KUKA KRL program: MyProgram_191().src

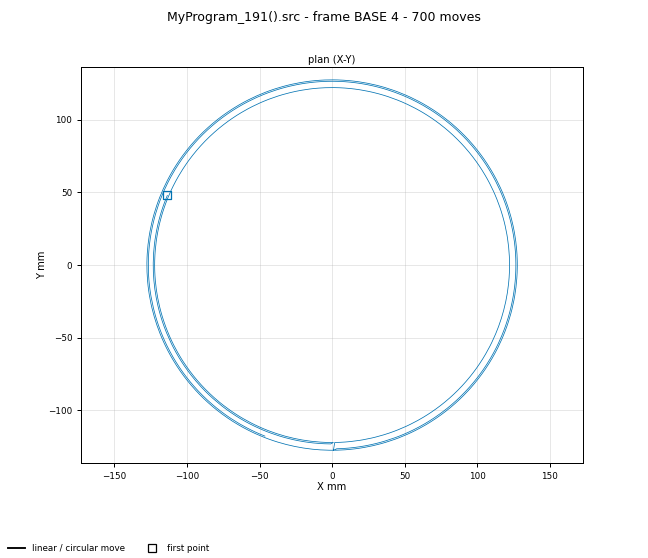
[picture p0: tool path of MyProgram_191().src in frame BASE 4, 700 of 700 moves have a stored position in this frame; points joined in program order, loops and branches not executed]
&ACCESS RVP
&REL 1
&PARAM TEMPLATE = C:\KRC\Roboter\Template\vorgabe
&PARAM EDITMASK = *
DEF MyProgram_191()
; ---- Setting reference (Base) ----
$BASE = BASE_DATA[4]

; --------------------------
; ---- Setting tool (TCP) ----
$TOOL = TOOL_DATA[3]
; --------------------------

$VEL.CP = VEL_APROX_PRINT
Startdeposition()
$VEL.CP = VEL_PRINT
LIN {X -113.4915,Y 47.9515,Z 138,A 153.5773,B 24.7784,C -1.6301,E1 24.6806,E2 292.6518} C_DIS
LIN {X -115.3064,Y 43.4036,Z 138,A 155.8653,B 24.7788,C -1.6235,E1 24.6783,E2 290.3668} C_DIS
LIN {X -116.411,Y 40.3471,Z 138,A 157.2234,B 24.7795,C -1.6121,E1 24.677,E2 289.0283} C_DIS
LIN {X -117.3905,Y 37.402,Z 138,A 158.8202,B 24.7794,C -1.6142,E1 24.6756,E2 287.4173} C_DIS
LIN {X -118.292,Y 34.4452,Z 138,A 160.3339,B 24.7794,C -1.6129,E1 24.6744,E2 285.8979} C_DIS
LIN {X -119.418,Y 30.3113,Z 138,A 162.2284,B 24.7801,C -1.6022,E1 24.6731,E2 284.0179} C_DIS
LIN {X -120.0632,Y 27.6462,Z 138,A 163.4846,B 24.7804,C -1.5973,E1 24.6723,E2 282.7662} C_DIS
LIN {X -120.9925,Y 23.2438,Z 138,A 165.6644,B 24.7806,C -1.5943,E1 24.6711,E2 280.5806} C_DIS
LIN {X -121.544,Y 20.1626,Z 138,A 167.1796,B 24.7806,C -1.5921,E1 24.6703,E2 279.0614} C_DIS
LIN {X -121.9177,Y 17.7672,Z 138,A 168.6693,B 24.78,C -1.6043,E1 24.6697,E2 277.5336} C_DIS
LIN {X -122.3545,Y 14.4523,Z 138,A 169.8773,B 24.7812,C -1.584,E1 24.6693,E2 276.3671} C_DIS
LIN {X -122.9178,Y 8.4272,Z 138,A 172.7848,B 24.7815,C -1.5788,E1 24.6687,E2 273.4544} C_DIS
LIN {X -123.1978,Y 1.4687,Z 138,A 176.8893,B 24.7798,C -1.6064,E1 24.6684,E2 269.2588} C_DIS
LIN {X -123.123,Y -4.5086,Z 138,A 178.5455,B 24.7833,C -1.5478,E1 24.6684,E2 267.7331} C_DIS
LIN {X -122.7454,Y -10.6368,Z 138,A -178.1412,B 24.7827,C -1.5585,E1 24.6691,E2 264.3741} C_DIS
LIN {X -122.0579,Y -16.7856,Z 138,A -175.5309,B 24.7839,C -1.5375,E1 24.67,E2 261.7985} C_DIS
LIN {X -121.0796,Y -22.7885,Z 138,A -172.5431,B 24.784,C -1.5354,E1 24.6714,E2 258.7978} C_DIS
LIN {X -120.0299,Y -27.7922,Z 138,A -170.1361,B 24.7844,C -1.5292,E1 24.6728,E2 256.3914} C_DIS
LIN {X -119.0923,Y -31.5671,Z 138,A -168.3681,B 24.7848,C -1.5218,E1 24.674,E2 254.6308} C_DIS
LIN {X -118.1261,Y -35.0118,Z 138,A -166.593,B 24.7848,C -1.5215,E1 24.6754,E2 252.8459} C_DIS
LIN {X -116.8426,Y -39.0802,Z 138,A -164.6565,B 24.7853,C -1.5134,E1 24.6771,E2 250.9178} C_DIS
LIN {X -115.6373,Y -42.5202,Z 138,A -163.0507,B 24.7858,C -1.5043,E1 24.6786,E2 249.3246} C_DIS
LIN {X -114.0487,Y -46.6116,Z 138,A -160.8655,B 24.7858,C -1.5046,E1 24.6809,E2 247.1262} C_DIS
LIN {X -110.5691,Y -54.3497,Z 138,A -156.9917,B 24.7866,C -1.49,E1 24.6854,E2 243.2662} C_DIS
LIN {X -109.2872,Y -56.8848,Z 138,A -155.6817,B 24.7869,C -1.4858,E1 24.687,E2 241.9592} C_DIS
LIN {X -107.5667,Y -60.078,Z 138,A -153.8305,B 24.7867,C -1.4884,E1 24.6895,E2 240.0919} C_DIS
LIN {X -105.3974,Y -63.8062,Z 138,A -152.0984,B 24.7877,C -1.4708,E1 24.692,E2 238.393} C_DIS
LIN {X -103.7402,Y -66.4666,Z 138,A -150.4231,B 24.7874,C -1.4766,E1 24.6945,E2 236.6952} C_DIS
LIN {X -101.5509,Y -69.7657,Z 138,A -148.5357,B 24.7875,C -1.4739,E1 24.6974,E2 234.8047} C_DIS
LIN {X -99.0053,Y -73.3341,Z 138,A -146.4687,B 24.7878,C -1.4701,E1 24.7008,E2 232.7369} C_DIS
LIN {X -96.9671,Y -76.0082,Z 138,A -144.6849,B 24.7874,C -1.4762,E1 24.7039,E2 230.93} C_DIS
LIN {X -93.5662,Y -80.158,Z 138,A -141.7973,B 24.7868,C -1.4881,E1 24.7093,E2 228.0006} C_DIS
LIN {X -90.2518,Y -83.8717,Z 138,A -140.0763,B 24.7885,C -1.4559,E1 24.7124,E2 226.3491} C_DIS
LIN {X -87.3058,Y -86.9342,Z 138,A -138.1334,B 24.7889,C -1.45,E1 24.7161,E2 224.4117} C_DIS
LIN {X -85.0375,Y -89.1542,Z 138,A -136.2104,B 24.7879,C -1.4673,E1 24.7201,E2 222.4395} C_DIS
LIN {X -82.0921,Y -91.8735,Z 138,A -135.1222,B 24.7901,C -1.4282,E1 24.7222,E2 221.4404} C_DIS
LIN {X -75.7976,Y -97.1325,Z 138,A -130.8704,B 24.7894,C -1.4406,E1 24.7315,E2 217.1426} C_DIS
LIN {X -72.8597,Y -99.3545,Z 138,A -129.1934,B 24.7896,C -1.4359,E1 24.7352,E2 215.4709} C_DIS
LIN {X -70.0805,Y -101.3345,Z 138,A -127.5112,B 24.7896,C -1.4376,E1 24.7391,E2 213.7788} C_DIS
LIN {X -66.1672,Y -103.9319,Z 138,A -125.6448,B 24.7905,C -1.4195,E1 24.7433,E2 211.9495} C_DIS
LIN {X -63.3912,Y -105.6482,Z 138,A -123.8429,B 24.7899,C -1.4303,E1 24.7477,E2 210.1162} C_DIS
LIN {X -59.6375,Y -107.811,Z 138,A -122.016,B 24.7906,C -1.4188,E1 24.7521,E2 208.3115} C_DIS
LIN {X -56.4456,Y -109.5155,Z 138,A -120.1657,B 24.7903,C -1.4243,E1 24.7567,E2 206.4429} C_DIS
LIN {X -53.2178,Y -111.1182,Z 138,A -118.5914,B 24.7906,C -1.4176,E1 24.7606,E2 204.8805} C_DIS
LIN {X -50.3384,Y -112.4519,Z 138,A -117.31,B 24.7912,C -1.4069,E1 24.7638,E2 203.6216} C_DIS
LIN {X -47.6999,Y -113.5965,Z 138,A -115.7642,B 24.7908,C -1.4151,E1 24.7679,E2 202.0525} C_DIS
LIN {X -45.0765,Y -114.6636,Z 138,A -114.595,B 24.7912,C -1.4069,E1 24.7709,E2 200.9003} C_DIS
LIN {X -41.9523,Y -115.8423,Z 138,A -113.0237,B 24.7912,C -1.4063,E1 24.775,E2 199.3272} C_DIS
LIN {X -39.061,Y -116.8489,Z 138,A -111.458,B 24.7909,C -1.4117,E1 24.7791,E2 197.7455} C_DIS
LIN {X -36.1486,Y -117.7825,Z 138,A -109.6372,B 24.79,C -1.4294,E1 24.7841,E2 195.8793} C_DIS
LIN {X -32.6362,Y -118.805,Z 138,A -108.2069,B 24.7907,C -1.4154,E1 24.7879,E2 194.48} C_DIS
LIN {X -26.8313,Y -120.2494,Z 138,A -105.5859,B 24.7912,C -1.4063,E1 24.795,E2 191.8771} C_DIS
LIN {X -23.219,Y -120.9973,Z 138,A -103.7988,B 24.7911,C -1.409,E1 24.7999,E2 190.0816} C_DIS
LIN {X -19.2814,Y -121.6877,Z 138,A -101.9432,B 24.7911,C -1.4083,E1 24.805,E2 188.226} C_DIS
LIN {X -16.1409,Y -122.1432,Z 138,A -100.6058,B 24.7915,C -1.4014,E1 24.8086,E2 186.904} C_DIS
LIN {X -13.0646,Y -122.5105,Z 138,A -98.9585,B 24.791,C -1.411,E1 24.8133,E2 185.2327} C_DIS
LIN {X -8.9867,Y -122.8769,Z 138,A -97.1257,B 24.7912,C -1.4075,E1 24.8184,E2 183.4074} C_DIS
LIN {X -5.1763,Y -123.097,Z 138,A -95.2835,B 24.791,C -1.4109,E1 24.8235,E2 181.5568} C_DIS
LIN {X -0.9339,Y -123.2019,Z 138,A -93.3832,B 24.7912,C -1.4077,E1 24.8288,E2 179.6639} C_DIS
LIN {X -0.9339,Y -123.2019,Z 138,A -93.3832,B 24.7912,C -1.4077,E1 24.8288,E2 179.6639} C_DIS
Enddeposition()
LIN {X 0.852,Y -122.218,Z 138,A -92.7365,B 24.3643,C -1.3273,E1 24.3999,E2 179.1497} C_DIS
Startdeposition()
$VEL.CP = VEL_PRINT
LIN {X -1.1747,Y -122.2187,Z 138,A -94.1532,B 24.3654,C -1.3055,E1 24.3958,E2 180.6191} C_DIS
LIN {X -4.4974,Y -122.1408,Z 138,A -95.7044,B 24.3654,C -1.3056,E1 24.3915,E2 182.1703} C_DIS
LIN {X -7.8683,Y -121.9703,Z 138,A -97.3656,B 24.3656,C -1.302,E1 24.3868,E2 183.8409} C_DIS
LIN {X -11.9845,Y -121.6346,Z 138,A -99.14,B 24.3652,C -1.3095,E1 24.3819,E2 185.598} C_DIS
LIN {X -14.6363,Y -121.3438,Z 138,A -100.3954,B 24.3652,C -1.3095,E1 24.3785,E2 186.8543} C_DIS
LIN {X -17.9306,Y -120.9025,Z 138,A -101.9314,B 24.3652,C -1.3108,E1 24.3742,E2 188.3883} C_DIS
LIN {X -20.5158,Y -120.4897,Z 138,A -103.2501,B 24.3654,C -1.307,E1 24.3706,E2 189.7174} C_DIS
LIN {X -23.5259,Y -119.939,Z 138,A -104.6142,B 24.3652,C -1.3108,E1 24.3668,E2 191.0739} C_DIS
LIN {X -26.0749,Y -119.4096,Z 138,A -105.9945,B 24.3655,C -1.3041,E1 24.363,E2 192.4721} C_DIS
LIN {X -29.708,Y -118.5582,Z 138,A -107.5972,B 24.3651,C -1.3117,E1 24.3587,E2 194.0587} C_DIS
LIN {X -32.2815,Y -117.8847,Z 138,A -108.8072,B 24.365,C -1.3141,E1 24.3555,E2 195.2647} C_DIS
LIN {X -35.4897,Y -116.9573,Z 138,A -110.2924,B 24.3648,C -1.3188,E1 24.3515,E2 196.7409} C_DIS
LIN {X -38.3454,Y -116.0524,Z 138,A -111.8191,B 24.365,C -1.3144,E1 24.3474,E2 198.2812} C_DIS
LIN {X -40.8707,Y -115.1886,Z 138,A -113.1758,B 24.3652,C -1.3108,E1 24.3438,E2 199.6495} C_DIS
LIN {X -43.6803,Y -114.1529,Z 138,A -114.5842,B 24.3652,C -1.3119,E1 24.3401,E2 201.0582} C_DIS
LIN {X -47.071,Y -112.7952,Z 138,A -116.2889,B 24.365,C -1.314,E1 24.3357,E2 202.7616} C_DIS
LIN {X -50.12,Y -111.474,Z 138,A -117.8196,B 24.3649,C -1.3169,E1 24.3318,E2 204.2891} C_DIS
LIN {X -53.3298,Y -109.9766,Z 138,A -119.4295,B 24.3646,C -1.3211,E1 24.3278,E2 205.893} C_DIS
LIN {X -56.0053,Y -108.6379,Z 138,A -120.8359,B 24.3646,C -1.3227,E1 24.3243,E2 207.2993} C_DIS
LIN {X -58.9088,Y -107.0922,Z 138,A -122.3786,B 24.3645,C -1.3248,E1 24.3205,E2 208.8415} C_DIS
LIN {X -61.2575,Y -105.7657,Z 138,A -123.7021,B 24.3645,C -1.324,E1 24.3173,E2 210.171} C_DIS
LIN {X -63.829,Y -104.234,Z 138,A -125.0526,B 24.3643,C -1.3284,E1 24.314,E2 211.515} C_DIS
LIN {X -66.6538,Y -102.4507,Z 138,A -126.6798,B 24.3643,C -1.3282,E1 24.3102,E2 213.1482} C_DIS
LIN {X -70.1137,Y -100.1153,Z 138,A -128.5919,B 24.364,C -1.3334,E1 24.3058,E2 215.0542} C_DIS
LIN {X -72.5492,Y -98.3643,Z 138,A -130.0014,B 24.3639,C -1.3357,E1 24.3026,E2 216.4632} C_DIS
LIN {X -74.9796,Y -96.5243,Z 138,A -131.4908,B 24.3639,C -1.3357,E1 24.2993,E2 217.9583} C_DIS
LIN {X -77.7047,Y -94.3448,Z 138,A -133.2287,B 24.3639,C -1.3342,E1 24.2955,E2 219.7062} C_DIS
LIN {X -81.0903,Y -91.4508,Z 138,A -135.2943,B 24.3637,C -1.3393,E1 24.2912,E2 221.7678} C_DIS
LIN {X -84.2804,Y -88.5197,Z 138,A -137.3634,B 24.3636,C -1.3419,E1 24.287,E2 223.8394} C_DIS
LIN {X -87.3611,Y -85.4805,Z 138,A -139.2827,B 24.3631,C -1.351,E1 24.2832,E2 225.7449} C_DIS
LIN {X -89.9719,Y -82.728,Z 138,A -141.1255,B 24.3631,C -1.3522,E1 24.2797,E2 227.5931} C_DIS
LIN {X -92.9374,Y -79.3826,Z 138,A -143.1994,B 24.3627,C -1.3579,E1 24.2759,E2 229.6626} C_DIS
LIN {X -95.4175,Y -76.3838,Z 138,A -145.1405,B 24.3627,C -1.3573,E1 24.2724,E2 231.6145} C_DIS
LIN {X -98.1723,Y -72.8088,Z 138,A -147.1088,B 24.3622,C -1.3688,E1 24.2691,E2 233.5645} C_DIS
LIN {X -100.0245,Y -70.2427,Z 138,A -148.764,B 24.3624,C -1.3652,E1 24.2664,E2 235.2367} C_DIS
LIN {X -102.4504,Y -66.6543,Z 138,A -150.5579,B 24.3615,C -1.3806,E1 24.2637,E2 237.0023} C_DIS
LIN {X -104.0513,Y -64.1269,Z 138,A -152.1971,B 24.3619,C -1.3742,E1 24.2612,E2 238.6658} C_DIS
LIN {X -106.3494,Y -60.2395,Z 138,A -154.1332,B 24.3612,C -1.3876,E1 24.2586,E2 240.5795} C_DIS
LIN {X -107.6369,Y -57.9065,Z 138,A -155.5184,B 24.3612,C -1.3853,E1 24.2567,E2 241.9778} C_DIS
LIN {X -109.0137,Y -55.2671,Z 138,A -156.8887,B 24.361,C -1.3903,E1 24.2549,E2 243.3435} C_DIS
LIN {X -110.5038,Y -52.2262,Z 138,A -158.4413,B 24.3607,C -1.3963,E1 24.2531,E2 244.8902} C_DIS
LIN {X -111.8809,Y -49.2103,Z 138,A -160.2288,B 24.361,C -1.3909,E1 24.251,E2 246.701} C_DIS
LIN {X -113.483,Y -45.3887,Z 138,A -161.957,B 24.3602,C -1.4057,E1 24.2492,E2 248.403} C_DIS
LIN {X -114.5655,Y -42.5825,Z 138,A -163.4393,B 24.3602,C -1.4068,E1 24.2477,E2 249.8911} C_DIS
LIN {X -115.9501,Y -38.6526,Z 138,A -165.4017,B 24.3598,C -1.4123,E1 24.2459,E2 251.8516} C_DIS
LIN {X -116.9523,Y -35.5062,Z 138,A -166.9,B 24.3595,C -1.4191,E1 24.2447,E2 253.3422} C_DIS
LIN {X -117.9764,Y -31.9412,Z 138,A -168.7779,B 24.3595,C -1.4186,E1 24.2433,E2 255.2325} C_DIS
LIN {X -118.839,Y -28.5616,Z 138,A -170.2955,B 24.3589,C -1.4286,E1 24.2423,E2 256.7347} C_DIS
LIN {X -119.5751,Y -25.3083,Z 138,A -171.8644,B 24.3587,C -1.4333,E1 24.2413,E2 258.3017} C_DIS
LIN {X -120.0655,Y -22.8641,Z 138,A -173.0773,B 24.3586,C -1.4351,E1 24.2407,E2 259.5175} C_DIS
LIN {X -120.6223,Y -19.7208,Z 138,A -174.5459,B 24.3583,C -1.441,E1 24.24,E2 260.9807} C_DIS
LIN {X -121.0678,Y -16.7739,Z 138,A -176.0325,B 24.3583,C -1.4417,E1 24.2394,E2 262.4747} C_DIS
LIN {X -121.4911,Y -13.3604,Z 138,A -177.4882,B 24.3576,C -1.4535,E1 24.2389,E2 263.9106} C_DIS
LIN {X -121.7522,Y -10.7287,Z 138,A -178.9175,B 24.3578,C -1.4496,E1 24.2386,E2 265.3584} C_DIS
LIN {X -121.9947,Y -7.4711,Z 138,A 179.6289,B 24.3573,C -1.4578,E1 24.2383,E2 266.801} C_DIS
LIN {X -122.1625,Y -3.8853,Z 138,A 177.7938,B 24.3573,C -1.4568,E1 24.2381,E2 268.6497} C_DIS
LIN {X -122.2263,Y -0.1231,Z 138,A 176.0896,B 24.3569,C -1.465,E1 24.2381,E2 270.3444} C_DIS
LIN {X -122.1899,Y 2.8995,Z 138,A 174.6031,B 24.3569,C -1.4668,E1 24.2381,E2 271.8359} C_DIS
LIN {X -122.0207,Y 7.0487,Z 138,A 172.7178,B 24.3563,C -1.4757,E1 24.2384,E2 273.7111} C_DIS
LIN {X -121.8016,Y 10.1449,Z 138,A 171.2313,B 24.3561,C -1.4792,E1 24.2387,E2 275.1983} C_DIS
LIN {X -121.4789,Y 13.4743,Z 138,A 169.764,B 24.3556,C -1.4885,E1 24.2391,E2 276.652} C_DIS
LIN {X -121.1532,Y 16.1393,Z 138,A 168.4248,B 24.3556,C -1.4892,E1 24.2396,E2 277.9977} C_DIS
LIN {X -120.599,Y 19.8602,Z 138,A 166.5949,B 24.3554,C -1.4922,E1 24.2404,E2 279.8315} C_DIS
LIN {X -119.9418,Y 23.5111,Z 138,A 164.9317,B 24.3549,C -1.5009,E1 24.2412,E2 281.4834} C_DIS
LIN {X -119.3249,Y 26.4675,Z 138,A 163.3914,B 24.3549,C -1.5003,E1 24.2421,E2 283.0346} C_DIS
LIN {X -118.5602,Y 29.6998,Z 138,A 161.7993,B 24.3547,C -1.5039,E1 24.2432,E2 284.6276} C_DIS
LIN {X -117.4803,Y 33.7233,Z 138,A 159.8547,B 24.3543,C -1.5104,E1 24.2446,E2 286.5679} C_DIS
LIN {X -116.6188,Y 36.5911,Z 138,A 158.4425,B 24.3541,C -1.5145,E1 24.2458,E2 287.9784} C_DIS
LIN {X -115.5784,Y 39.7513,Z 138,A 156.8856,B 24.3538,C -1.5196,E1 24.2472,E2 289.5321} C_DIS
LIN {X -114.3716,Y 43.1001,Z 138,A 155.1973,B 24.3535,C -1.524,E1 24.2488,E2 291.2195} C_DIS
LIN {X -113.0423,Y 46.4791,Z 138,A 153.48,B 24.3532,C -1.5286,E1 24.2506,E2 292.9354} C_DIS
LIN {X -111.8746,Y 49.2245,Z 138,A 152.0617,B 24.353,C -1.532,E1 24.2522,E2 294.3534} C_DIS
LIN {X -110.6278,Y 51.9657,Z 138,A 150.7478,B 24.3525,C -1.5404,E1 24.2537,E2 295.6543} C_DIS
LIN {X -109.3219,Y 54.6585,Z 138,A 149.3353,B 24.3523,C -1.5442,E1 24.2555,E2 297.0653} C_DIS
LIN {X -107.5634,Y 58.0433,Z 138,A 147.521,B 24.3521,C -1.5484,E1 24.2578,E2 298.8792} C_DIS
LIN {X -105.7031,Y 61.3657,Z 138,A 145.7038,B 24.3518,C -1.5523,E1 24.2603,E2 300.6967} C_DIS
LIN {X -104.2135,Y 63.8625,Z 138,A 144.4625,B 24.3513,C -1.5614,E1 24.2621,E2 301.9224} C_DIS
LIN {X -102.6967,Y 66.2749,Z 138,A 142.8668,B 24.3517,C -1.5542,E1 24.2645,E2 303.5438} C_DIS
LIN {X -100.1153,Y 70.1137,Z 138,A 140.8425,B 24.351,C -1.5664,E1 24.2677,E2 305.5489} C_DIS
LIN {X -98.3676,Y 72.5447,Z 138,A 139.3725,B 24.351,C -1.5674,E1 24.2701,E2 307.0236} C_DIS
LIN {X -95.8913,Y 75.7882,Z 138,A 137.3452,B 24.351,C -1.5678,E1 24.2736,E2 309.06} C_DIS
LIN {X -93.1416,Y 79.1423,Z 138,A 135.4038,B 24.3503,C -1.577,E1 24.277,E2 310.9882} C_DIS
LIN {X -90.5637,Y 82.0798,Z 138,A 133.4693,B 24.3503,C -1.5773,E1 24.2807,E2 312.9307} C_DIS
LIN {X -87.5282,Y 85.3101,Z 138,A 131.3586,B 24.3501,C -1.5811,E1 24.2847,E2 315.0416} C_DIS
LIN {X -84.2766,Y 88.5233,Z 138,A 129.2184,B 24.3498,C -1.5864,E1 24.289,E2 317.1782} C_DIS
LIN {X -81.09,Y 91.4512,Z 138,A 127.2157,B 24.3494,C -1.5922,E1 24.2932,E2 319.1749} C_DIS
LIN {X -78.0552,Y 94.0546,Z 138,A 125.3237,B 24.3492,C -1.5957,E1 24.2972,E2 321.066} C_DIS
LIN {X -74.6019,Y 96.8171,Z 138,A 123.2103,B 24.349,C -1.5984,E1 24.3018,E2 323.1806} C_DIS
LIN {X -71.6013,Y 99.0563,Z 138,A 121.6099,B 24.3484,C -1.6087,E1 24.3054,E2 324.7618} C_DIS
LIN {X -69.1523,Y 100.781,Z 138,A 120.1252,B 24.3484,C -1.6081,E1 24.3088,E2 326.2533} C_DIS
LIN {X -65.6572,Y 103.0926,Z 138,A 118.1515,B 24.3482,C -1.6115,E1 24.3134,E2 328.2253} C_DIS
LIN {X -62.8163,Y 104.8478,Z 138,A 116.7156,B 24.3477,C -1.62,E1 24.3168,E2 329.6451} C_DIS
LIN {X -60.2331,Y 106.3531,Z 138,A 115.2944,B 24.3476,C -1.6216,E1 24.3203,E2 331.0666} C_DIS
LIN {X -57.9016,Y 107.6396,Z 138,A 113.9157,B 24.3478,C -1.6181,E1 24.3237,E2 332.4578} C_DIS
LIN {X -54.9576,Y 109.1713,Z 138,A 112.4297,B 24.3475,C -1.6237,E1 24.3273,E2 333.9343} C_DIS
LIN {X -52.1843,Y 110.5239,Z 138,A 110.9805,B 24.3473,C -1.6259,E1 24.331,E2 335.3821} C_DIS
LIN {X -49.5255,Y 111.7399,Z 138,A 109.6064,B 24.3473,C -1.6278,E1 24.3345,E2 336.755} C_DIS
LIN {X -47.0747,Y 112.7936,Z 138,A 108.2983,B 24.3473,C -1.6272,E1 24.3379,E2 338.0678} C_DIS
LIN {X -43.5437,Y 114.2055,Z 138,A 106.3657,B 24.3475,C -1.623,E1 24.3429,E2 340.0147} C_DIS
LIN {X -39.8373,Y 115.5486,Z 138,A 104.7562,B 24.3467,C -1.6358,E1 24.3471,E2 341.5964} C_DIS
LIN {X -37.2178,Y 116.4185,Z 138,A 103.358,B 24.3469,C -1.6328,E1 24.3508,E2 343.0046} C_DIS
LIN {X -34.0409,Y 117.3872,Z 138,A 101.8572,B 24.3466,C -1.637,E1 24.3548,E2 344.4977} C_DIS
LIN {X -31.1552,Y 118.186,Z 138,A 100.4972,B 24.3464,C -1.6403,E1 24.3585,E2 345.8517} C_DIS
LIN {X -28.5721,Y 118.8365,Z 138,A 99.1492,B 24.3466,C -1.6372,E1 24.3621,E2 347.2093} C_DIS
LIN {X -25.0186,Y 119.6369,Z 138,A 97.3083,B 24.3469,C -1.6328,E1 24.3672,E2 349.0633} C_DIS
LIN {X -21.2072,Y 120.3696,Z 138,A 95.6706,B 24.3463,C -1.6422,E1 24.3716,E2 350.6798} C_DIS
LIN {X -18.2515,Y 120.8536,Z 138,A 94.2678,B 24.3463,C -1.6432,E1 24.3755,E2 352.0814} C_DIS
LIN {X -15.318,Y 121.2608,Z 138,A 92.7722,B 24.3465,C -1.6393,E1 24.3797,E2 353.5877} C_DIS
LIN {X -12.3074,Y 121.6036,Z 138,A 91.4293,B 24.3462,C -1.6435,E1 24.3834,E2 354.9211} C_DIS
LIN {X -8.9578,Y 121.8946,Z 138,A 89.8085,B 24.3462,C -1.6423,E1 24.3879,E2 356.5458} C_DIS
LIN {X -4.8186,Y 122.1283,Z 138,A 87.9232,B 24.3461,C -1.6455,E1 24.3931,E2 358.4236} C_DIS
LIN {X -1.8245,Y 122.2099,Z 138,A 86.4961,B 24.3461,C -1.6449,E1 24.3971,E2 359.8524} C_DIS
LIN {X 1.1685,Y 122.2188,Z 138,A 84.9591,B 24.3465,C -1.6391,E1 24.4015,E2 361.4034} C_DIS
LIN {X 5.2319,Y 122.1122,Z 138,A 83.0229,B 24.3465,C -1.6379,E1 24.4069,E2 363.342} C_DIS
LIN {X 8.669,Y 121.9156,Z 138,A 81.588,B 24.3461,C -1.6459,E1 24.4108,E2 364.7569} C_DIS
LIN {X 11.9806,Y 121.635,Z 138,A 80.0447,B 24.3461,C -1.6464,E1 24.4151,E2 366.298} C_DIS
LIN {X 15.5903,Y 121.2251,Z 138,A 78.2696,B 24.3463,C -1.6428,E1 24.42,E2 368.0805} C_DIS
LIN {X 19.4212,Y 120.6723,Z 138,A 76.5086,B 24.3461,C -1.6447,E1 24.4249,E2 369.8353} C_DIS
LIN {X 22.3721,Y 120.1595,Z 138,A 75.185,B 24.3459,C -1.6478,E1 24.4285,E2 371.1498} C_DIS
LIN {X 25.0145,Y 119.6377,Z 138,A 73.8644,B 24.3461,C -1.6446,E1 24.4321,E2 372.4765} C_DIS
LIN {X 28.1611,Y 118.9355,Z 138,A 72.171,B 24.3467,C -1.6354,E1 24.4368,E2 374.1897} C_DIS
LIN {X 32.2917,Y 117.8818,Z 138,A 70.3516,B 24.3463,C -1.6423,E1 24.4417,E2 375.9894} C_DIS
LIN {X 35.4859,Y 116.9585,Z 138,A 68.9156,B 24.346,C -1.6468,E1 24.4455,E2 377.412} C_DIS
LIN {X 38.6541,Y 115.9496,Z 138,A 67.1084,B 24.3468,C -1.6341,E1 24.4503,E2 379.2465} C_DIS
LIN {X 42.5823,Y 114.5656,Z 138,A 65.4196,B 24.3462,C -1.6445,E1 24.4547,E2 380.9067} C_DIS
LIN {X 45.0698,Y 113.6116,Z 138,A 63.8894,B 24.3471,C -1.6302,E1 24.4588,E2 382.468} C_DIS
LIN {X 48.3908,Y 112.2353,Z 138,A 62.3278,B 24.3468,C -1.6341,E1 24.4627,E2 384.0164} C_DIS
LIN {X 51.9751,Y 110.6235,Z 138,A 60.5174,B 24.3468,C -1.6333,E1 24.4673,E2 385.8238} C_DIS
LIN {X 54.6661,Y 109.3182,Z 138,A 59.1189,B 24.347,C -1.6317,E1 24.4708,E2 387.2223} C_DIS
LIN {X 57.3256,Y 107.9467,Z 138,A 57.6875,B 24.3472,C -1.6285,E1 24.4744,E2 388.6574} C_DIS
LIN {X 60.2381,Y 106.3503,Z 138,A 56.221,B 24.347,C -1.6305,E1 24.4779,E2 390.1146} C_DIS
LIN {X 62.8397,Y 104.8338,Z 138,A 54.7644,B 24.3473,C -1.6263,E1 24.4815,E2 391.5768} C_DIS
LIN {X 65.6974,Y 103.0668,Z 138,A 53.056,B 24.3478,C -1.6176,E1 24.4855,E2 393.3007} C_DIS
LIN {X 68.8222,Y 101.0074,Z 138,A 51.4364,B 24.3476,C -1.621,E1 24.4893,E2 394.9065} C_DIS
LIN {X 71.3331,Y 99.2499,Z 138,A 50.1139,B 24.3474,C -1.6239,E1 24.4923,E2 396.2172} C_DIS
LIN {X 74.0069,Y 97.2725,Z 138,A 48.3132,B 24.3483,C -1.6097,E1 24.4963,E2 398.0456} C_DIS
LIN {X 77.5317,Y 94.4868,Z 138,A 46.3116,B 24.3483,C -1.6107,E1 24.5007,E2 400.0371} C_DIS
LIN {X 80.2808,Y 92.1622,Z 138,A 44.6537,B 24.3483,C -1.6088,E1 24.5042,E2 401.693} C_DIS
LIN {X 83.1858,Y 89.5489,Z 138,A 42.7529,B 24.3488,C -1.6017,E1 24.5081,E2 403.6028} C_DIS
LIN {X 86.088,Y 86.7625,Z 138,A 40.861,B 24.3491,C -1.5974,E1 24.5119,E2 405.4971} C_DIS
LIN {X 89.0365,Y 83.7341,Z 138,A 38.891,B 24.3493,C -1.5936,E1 24.5157,E2 407.4677} C_DIS
LIN {X 91.559,Y 80.9679,Z 138,A 37.1512,B 24.3495,C -1.5903,E1 24.519,E2 409.2075} C_DIS
LIN {X 94.3821,Y 77.6597,Z 138,A 35.2027,B 24.3495,C -1.5897,E1 24.5224,E2 411.148} C_DIS
LIN {X 96.8164,Y 74.6028,Z 138,A 33.3331,B 24.35,C -1.5834,E1 24.5257,E2 413.0237} C_DIS
LIN {X 99.0689,Y 71.5838,Z 138,A 31.608,B 24.3501,C -1.581,E1 24.5285,E2 414.7463} C_DIS
LIN {X 101.4348,Y 68.1908,Z 138,A 29.6468,B 24.3505,C -1.5749,E1 24.5316,E2 416.7123} C_DIS
LIN {X 103.1672,Y 65.5402,Z 138,A 28.1069,B 24.3509,C -1.5683,E1 24.534,E2 418.2601} C_DIS
LIN {X 105.4236,Y 61.8444,Z 138,A 26.1818,B 24.3509,C -1.5679,E1 24.5367,E2 420.176} C_DIS
LIN {X 106.9194,Y 59.2208,Z 138,A 24.8348,B 24.3509,C -1.5673,E1 24.5386,E2 421.5173} C_DIS
LIN {X 108.489,Y 56.2929,Z 138,A 23.2787,B 24.3512,C -1.563,E1 24.5406,E2 423.0752} C_DIS
LIN {X 109.8352,Y 53.6181,Z 138,A 21.8856,B 24.3514,C -1.5596,E1 24.5423,E2 424.469} C_DIS
LIN {X 111.0995,Y 50.9457,Z 138,A 20.5469,B 24.3514,C -1.5579,E1 24.5439,E2 425.8044} C_DIS
LIN {X 112.1692,Y 48.5437,Z 138,A 19.2668,B 24.3519,C -1.552,E1 24.5453,E2 427.0914} C_DIS
LIN {X 113.4868,Y 45.3792,Z 138,A 17.6905,B 24.352,C -1.5488,E1 24.547,E2 428.6667} C_DIS
LIN {X 114.565,Y 42.5839,Z 138,A 16.3492,B 24.3521,C -1.5477,E1 24.5483,E2 430.003} C_DIS
LIN {X 115.5744,Y 39.7629,Z 138,A 14.9561,B 24.3523,C -1.544,E1 24.5496,E2 431.3969} C_DIS
LIN {X 116.4249,Y 37.198,Z 138,A 13.5879,B 24.3529,C -1.5352,E1 24.5508,E2 432.7783} C_DIS
LIN {X 117.3902,Y 34.0308,Z 138,A 11.9691,B 24.3533,C -1.5272,E1 24.5521,E2 434.4069} C_DIS
LIN {X 118.479,Y 30.0198,Z 138,A 10.1674,B 24.3533,C -1.5283,E1 24.5534,E2 436.1953} C_DIS
LIN {X 119.1774,Y 27.1152,Z 138,A 8.7309,B 24.3536,C -1.5221,E1 24.5543,E2 437.6381} C_DIS
LIN {X 119.8759,Y 23.8439,Z 138,A 7.2256,B 24.3537,C -1.5202,E1 24.5552,E2 439.139} C_DIS
LIN {X 120.3669,Y 21.2227,Z 138,A 5.9821,B 24.3539,C -1.5166,E1 24.5558,E2 440.3837} C_DIS
LIN {X 120.8017,Y 18.5867,Z 138,A 4.7116,B 24.3542,C -1.5117,E1 24.5563,E2 441.6583} C_DIS
LIN {X 121.3054,Y 14.9578,Z 138,A 3.0159,B 24.3545,C -1.5073,E1 24.557,E2 443.3544} C_DIS
LIN {X 121.6036,Y 12.3073,Z 138,A 1.7691,B 24.3547,C -1.5034,E1 24.5573,E2 444.603} C_DIS
LIN {X 121.8918,Y 8.9951,Z 138,A 0.3033,B 24.3547,C -1.5029,E1 24.5577,E2 446.061} C_DIS
LIN {X 122.0729,Y 6.0625,Z 138,A -1.1822,B 24.3553,C -1.4931,E1 24.5579,E2 447.561} C_DIS
LIN {X 122.2099,Y 1.827,Z 138,A -3.0667,B 24.3553,C -1.4917,E1 24.558,E2 449.4375} C_DIS
LIN {X 122.2153,Y -1.4969,Z 138,A -4.6683,B 24.3558,C -1.4844,E1 24.558,E2 451.0468} C_DIS
LIN {X 122.1283,Y -4.8191,Z 138,A -6.2088,B 24.356,C -1.4802,E1 24.5579,E2 452.588} C_DIS
LIN {X 121.9159,Y -8.6657,Z 138,A -8.0616,B 24.3565,C -1.472,E1 24.5576,E2 454.4494} C_DIS
LIN {X 121.5558,Y -12.7597,Z 138,A -9.9936,B 24.3569,C -1.4654,E1 24.557,E2 456.3854} C_DIS
LIN {X 121.156,Y -16.1174,Z 138,A -11.506,B 24.3569,C -1.4638,E1 24.5565,E2 457.8925} C_DIS
LIN {X 120.7332,Y -19.029,Z 138,A -12.8222,B 24.3571,C -1.4624,E1 24.556,E2 459.2041} C_DIS
LIN {X 120.1584,Y -22.3784,Z 138,A -14.3591,B 24.3571,C -1.46,E1 24.5552,E2 460.7377} C_DIS
LIN {X 119.6367,Y -25.0196,Z 138,A -15.6741,B 24.3576,C -1.4533,E1 24.5545,E2 462.0609} C_DIS
LIN {X 118.9142,Y -28.2497,Z 138,A -17.226,B 24.3579,C -1.4483,E1 24.5535,E2 463.6156} C_DIS
LIN {X 118.187,Y -31.1516,Z 138,A -18.4902,B 24.3577,C -1.4505,E1 24.5526,E2 464.8668} C_DIS
LIN {X 117.4819,Y -33.7176,Z 138,A -19.9614,B 24.3586,C -1.4356,E1 24.5515,E2 466.3655} C_DIS
LIN {X 116.6226,Y -36.579,Z 138,A -21.3566,B 24.3588,C -1.4314,E1 24.5504,E2 467.7627} C_DIS
LIN {X 115.5762,Y -39.7575,Z 138,A -22.6783,B 24.3584,C -1.4385,E1 24.5492,E2 469.0595} C_DIS
LIN {X 114.6008,Y -42.4884,Z 138,A -24.0658,B 24.3587,C -1.4329,E1 24.5479,E2 470.4526} C_DIS
LIN {X 113.6089,Y -45.0766,Z 138,A -25.4399,B 24.3591,C -1.4251,E1 24.5465,E2 471.8375} C_DIS
LIN {X 112.6264,Y -47.4751,Z 138,A -26.7235,B 24.3595,C -1.418,E1 24.5451,E2 473.131} C_DIS
LIN {X 111.1086,Y -50.9259,Z 138,A -28.2644,B 24.3592,C -1.4237,E1 24.5434,E2 474.6497} C_DIS
LIN {X 109.9776,Y -53.3277,Z 138,A -29.6473,B 24.3598,C -1.4131,E1 24.5417,E2 476.0504} C_DIS
LIN {X 108.6491,Y -55.9834,Z 138,A -31.033,B 24.36,C -1.4092,E1 24.5399,E2 477.4378} C_DIS
LIN {X 107.075,Y -58.9399,Z 138,A -32.5812,B 24.3602,C -1.4056,E1 24.5379,E2 478.9864} C_DIS
LIN {X 105.7622,Y -61.2636,Z 138,A -33.8873,B 24.3605,C -1.3992,E1 24.5361,E2 480.3009} C_DIS
LIN {X 103.7135,Y -64.6714,Z 138,A -35.7592,B 24.3609,C -1.3934,E1 24.5333,E2 482.177} C_DIS
LIN {X 101.4374,Y -68.187,Z 138,A -37.8095,B 24.3614,C -1.3836,E1 24.5302,E2 484.2405} C_DIS
LIN {X 99.2488,Y -71.3346,Z 138,A -39.4241,B 24.3612,C -1.3875,E1 24.5276,E2 485.8378} C_DIS
LIN {X 97.273,Y -74.0063,Z 138,A -41.0994,B 24.3617,C -1.3775,E1 24.5247,E2 487.5288} C_DIS
LIN {X 94.8419,Y -77.0972,Z 138,A -42.9286,B 24.3619,C -1.3732,E1 24.5215,E2 489.3596} C_DIS
LIN {X 92.163,Y -80.2798,Z 138,A -44.7745,B 24.3619,C -1.3732,E1 24.5182,E2 491.197} C_DIS
LIN {X 89.551,Y -83.1836,Z 138,A -46.6766,B 24.3624,C -1.365,E1 24.5146,E2 493.1102} C_DIS
LIN {X 86.5318,Y -86.3202,Z 138,A -48.6545,B 24.3624,C -1.363,E1 24.5108,E2 495.0842} C_DIS
LIN {X 83.7307,Y -89.0397,Z 138,A -50.5354,B 24.3628,C -1.3561,E1 24.5069,E2 496.9738} C_DIS
LIN {X 80.966,Y -91.5608,Z 138,A -52.2747,B 24.363,C -1.3527,E1 24.5033,E2 498.7141} C_DIS
LIN {X 77.6568,Y -94.3845,Z 138,A -54.2242,B 24.363,C -1.3523,E1 24.4992,E2 500.6567} C_DIS
LIN {X 74.6009,Y -96.8178,Z 138,A -56.1703,B 24.3635,C -1.3428,E1 24.4949,E2 502.6184} C_DIS
LIN {X 71.6009,Y -99.0566,Z 138,A -57.81,B 24.3635,C -1.3446,E1 24.4912,E2 504.2477} C_DIS
LIN {X 68.1881,Y -101.4367,Z 138,A -59.7848,B 24.3637,C -1.3395,E1 24.4866,E2 506.228} C_DIS
LIN {X 65.6646,Y -103.0879,Z 138,A -61.0446,B 24.3635,C -1.3441,E1 24.4837,E2 507.4725} C_DIS
LIN {X 62.8335,Y -104.8375,Z 138,A -62.8091,B 24.3641,C -1.3314,E1 24.4795,E2 509.262} C_DIS
LIN {X 59.0212,Y -107.03,Z 138,A -64.6958,B 24.3639,C -1.336,E1 24.4749,E2 511.1318} C_DIS
LIN {X 56.2496,Y -108.5118,Z 138,A -66.1484,B 24.3639,C -1.3344,E1 24.4713,E2 512.584} C_DIS
LIN {X 53.928,Y -109.6823,Z 138,A -67.4464,B 24.3643,C -1.3287,E1 24.468,E2 513.8923} C_DIS
LIN {X 50.888,Y -111.1262,Z 138,A -68.9691,B 24.3643,C -1.3287,E1 24.4642,E2 515.4107} C_DIS
LIN {X 48.1495,Y -112.3396,Z 138,A -70.3222,B 24.3643,C -1.3291,E1 24.4608,E2 516.7597} C_DIS
LIN {X 45.3817,Y -113.4859,Z 138,A -71.7661,B 24.3644,C -1.3252,E1 24.457,E2 518.2097} C_DIS
LIN {X 42.7791,Y -114.4919,Z 138,A -73.104,B 24.3646,C -1.322,E1 24.4535,E2 519.5524} C_DIS
LIN {X 39.3734,Y -115.7094,Z 138,A -74.9712,B 24.3651,C -1.3117,E1 24.4485,E2 521.4406} C_DIS
LIN {X 35.4629,Y -116.9655,Z 138,A -76.6286,B 24.3646,C -1.322,E1 24.4442,E2 523.0699} C_DIS
LIN {X 32.5932,Y -117.7975,Z 138,A -78.0746,B 24.3648,C -1.3183,E1 24.4403,E2 524.5223} C_DIS
LIN {X 30.022,Y -118.4785,Z 138,A -79.3196,B 24.3648,C -1.3171,E1 24.4369,E2 525.7683} C_DIS
LIN {X 27.1194,Y -119.1764,Z 138,A -80.7621,B 24.365,C -1.3137,E1 24.433,E2 527.2169} C_DIS
LIN {X 23.841,Y -119.8765,Z 138,A -82.2781,B 24.365,C -1.3149,E1 24.4288,E2 528.7281} C_DIS
LIN {X 21.2194,Y -120.3674,Z 138,A -83.4918,B 24.365,C -1.3156,E1 24.4255,E2 529.9387} C_DIS
LIN {X 18.6654,Y -120.7895,Z 138,A -84.8042,B 24.3652,C -1.3101,E1 24.4219,E2 531.2631} C_DIS
LIN {X 14.955,Y -121.3057,Z 138,A -86.51,B 24.3652,C -1.3113,E1 24.4171,E2 532.9646} C_DIS
LIN {X 12.3037,Y -121.604,Z 138,A -87.7649,B 24.3652,C -1.3104,E1 24.4137,E2 534.2208} C_DIS
LIN {X 8.9925,Y -121.892,Z 138,A -89.3062,B 24.3652,C -1.3104,E1 24.4094,E2 535.7612} C_DIS
LIN {X 5.7189,Y -122.0901,Z 138,A -90.9883,B 24.3656,C -1.3031,E1 24.4046,E2 537.4604} C_DIS
LIN {X 1.8206,Y -122.21,Z 138,A -92.6906,B 24.3653,C -1.3084,E1 24.3999,E2 539.1497} C_DIS
LIN {X 1.8206,Y -122.21,Z 138,A -92.6906,B 24.3653,C -1.3084,E1 24.3999,E2 539.1497} C_DIS
Enddeposition()
LIN {X 0.903,Y -127.5582,Z 139,A -92.8335,B 24.9653,C -1.3615,E1 25.0014,E2 539.248} C_DIS
Startdeposition()
$VEL.CP = VEL_PRINT
LIN {X -1.9731,Y -127.547,Z 139,A -94.4529,B 24.9661,C -1.3449,E1 24.9968,E2 540.9066} C_DIS
LIN {X -5.6447,Y -127.439,Z 139,A -96.0438,B 24.966,C -1.3476,E1 24.9924,E2 542.4915} C_DIS
LIN {X -8.0273,Y -127.3094,Z 139,A -97.1271,B 24.966,C -1.347,E1 24.9893,E2 543.5765} C_DIS
LIN {X -11.3552,Y -127.0572,Z 139,A -98.6178,B 24.966,C -1.3474,E1 24.9852,E2 545.0668} C_DIS
LIN {X -13.6413,Y -126.8306,Z 139,A -99.6888,B 24.966,C -1.3456,E1 24.9822,E2 546.1427} C_DIS
LIN {X -17.3099,Y -126.3843,Z 139,A -101.3219,B 24.966,C -1.3472,E1 24.9777,E2 547.7732} C_DIS
LIN {X -19.649,Y -126.0396,Z 139,A -102.3823,B 24.966,C -1.3476,E1 24.9747,E2 548.8336} C_DIS
LIN {X -22.9388,Y -125.4834,Z 139,A -103.864,B 24.966,C -1.349,E1 24.9707,E2 550.3136} C_DIS
LIN {X -25.5944,Y -124.968,Z 139,A -105.1454,B 24.966,C -1.3462,E1 24.9671,E2 551.6029} C_DIS
LIN {X -28.8598,Y -124.2552,Z 139,A -106.6046,B 24.966,C -1.349,E1 24.9632,E2 553.0574} C_DIS
LIN {X -31.6241,Y -123.58,Z 139,A -107.9241,B 24.966,C -1.3477,E1 24.9596,E2 554.3818} C_DIS
LIN {X -34.719,Y -122.7467,Z 139,A -109.3669,B 24.966,C -1.3485,E1 24.9557,E2 555.8249} C_DIS
LIN {X -37.6032,Y -121.8938,Z 139,A -110.7401,B 24.966,C -1.3485,E1 24.952,E2 557.2007} C_DIS
LIN {X -40.6766,Y -120.9032,Z 139,A -112.1312,B 24.9657,C -1.3525,E1 24.9484,E2 558.5848} C_DIS
LIN {X -43.9471,Y -119.7546,Z 139,A -113.6986,B 24.9657,C -1.3533,E1 24.9442,E2 560.1533} C_DIS
LIN {X -46.7222,Y -118.6984,Z 139,A -115.0406,B 24.9657,C -1.3542,E1 24.9407,E2 561.496} C_DIS
LIN {X -49.8926,Y -117.4025,Z 139,A -116.5901,B 24.9656,C -1.3553,E1 24.9367,E2 563.0465} C_DIS
LIN {X -52.3927,Y -116.3061,Z 139,A -117.8623,B 24.9656,C -1.3545,E1 24.9335,E2 564.3237} C_DIS
LIN {X -55.3841,Y -114.912,Z 139,A -119.3328,B 24.9656,C -1.3568,E1 24.9298,E2 565.7923} C_DIS
LIN {X -58.1516,Y -113.5362,Z 139,A -120.748,B 24.9655,C -1.3573,E1 24.9262,E2 567.2101} C_DIS
LIN {X -61.2316,Y -111.907,Z 139,A -122.3187,B 24.9654,C -1.3591,E1 24.9224,E2 568.7809} C_DIS
LIN {X -64.9415,Y -109.7961,Z 139,A -124.3255,B 24.9654,C -1.3576,E1 24.9175,E2 570.7973} C_DIS
LIN {X -68.5598,Y -107.5736,Z 139,A -126.2373,B 24.9654,C -1.3604,E1 24.913,E2 572.7086} C_DIS
LIN {X -71.8444,Y -105.4087,Z 139,A -128.0285,B 24.9652,C -1.3621,E1 24.9088,E2 574.5016} C_DIS
LIN {X -75.3495,Y -102.9317,Z 139,A -129.9343,B 24.965,C -1.3665,E1 24.9045,E2 576.4036} C_DIS
LIN {X -78.9255,Y -100.216,Z 139,A -131.8818,B 24.9647,C -1.3735,E1 24.9002,E2 578.3416} C_DIS
LIN {X -82.0849,Y -97.645,Z 139,A -133.7275,B 24.9645,C -1.3762,E1 24.8963,E2 580.1878} C_DIS
LIN {X -85.2676,Y -94.8785,Z 139,A -135.6134,B 24.9643,C -1.3804,E1 24.8923,E2 582.0712} C_DIS
LIN {X -88.2756,Y -92.0864,Z 139,A -137.5329,B 24.9643,C -1.3807,E1 24.8884,E2 583.9979} C_DIS
LIN {X -91.3615,Y -89.0264,Z 139,A -139.5449,B 24.9643,C -1.3821,E1 24.8844,E2 586.0151} C_DIS
LIN {X -94.1934,Y -86.0245,Z 139,A -141.3132,B 24.9638,C -1.3903,E1 24.8811,E2 587.7717} C_DIS
LIN {X -96.9248,Y -82.9349,Z 139,A -143.2647,B 24.9638,C -1.39,E1 24.8775,E2 589.7329} C_DIS
LIN {X -99.6688,Y -79.6155,Z 139,A -145.1771,B 24.9635,C -1.3957,E1 24.8741,E2 591.6406} C_DIS
LIN {X -102.0704,Y -76.5131,Z 139,A -146.9654,B 24.9633,C -1.3988,E1 24.8711,E2 593.4299} C_DIS
LIN {X -104.6065,Y -73.0066,Z 139,A -148.8997,B 24.9631,C -1.4042,E1 24.868,E2 595.3608} C_DIS
LIN {X -107.1425,Y -69.2316,Z 139,A -150.8614,B 24.9626,C -1.4133,E1 24.865,E2 597.3107} C_DIS
LIN {X -109.2523,Y -65.8515,Z 139,A -152.7335,B 24.9626,C -1.4143,E1 24.8622,E2 599.19} C_DIS
LIN {X -111.3893,Y -62.1694,Z 139,A -154.5681,B 24.9621,C -1.4231,E1 24.8597,E2 601.0132} C_DIS
LIN {X -113.0758,Y -59.0417,Z 139,A -156.2154,B 24.9619,C -1.4253,E1 24.8576,E2 602.6642} C_DIS
LIN {X -114.5646,Y -56.0988,Z 139,A -157.6951,B 24.9617,C -1.4296,E1 24.8557,E2 604.1416} C_DIS
LIN {X -115.9552,Y -53.1653,Z 139,A -159.1521,B 24.9615,C -1.4338,E1 24.854,E2 605.5964} C_DIS
LIN {X -117.2631,Y -50.2149,Z 139,A -160.5637,B 24.9612,C -1.4398,E1 24.8524,E2 607.0016} C_DIS
LIN {X -118.4936,Y -47.2388,Z 139,A -162.0207,B 24.961,C -1.4436,E1 24.8509,E2 608.4576} C_DIS
LIN {X -119.7175,Y -44.0486,Z 139,A -163.5685,B 24.9607,C -1.4476,E1 24.8494,E2 610.0046} C_DIS
LIN {X -120.6116,Y -41.5322,Z 139,A -164.8324,B 24.9607,C -1.4483,E1 24.8482,E2 611.274} C_DIS
LIN {X -121.7188,Y -38.1708,Z 139,A -166.3622,B 24.9603,C -1.4559,E1 24.8469,E2 612.7945} C_DIS
LIN {X -122.4508,Y -35.7468,Z 139,A -167.5359,B 24.9602,C -1.4577,E1 24.846,E2 613.9705} C_DIS
LIN {X -123.3005,Y -32.6963,Z 139,A -168.9671,B 24.96,C -1.4618,E1 24.8449,E2 615.4005} C_DIS
LIN {X -124.0494,Y -29.7291,Z 139,A -170.3896,B 24.9599,C -1.4639,E1 24.844,E2 616.8263} C_DIS
LIN {X -124.7413,Y -26.6777,Z 139,A -171.8015,B 24.9596,C -1.468,E1 24.8431,E2 618.2366} C_DIS
LIN {X -125.393,Y -23.429,Z 139,A -173.2195,B 24.9592,C -1.4759,E1 24.8424,E2 619.6441} C_DIS
LIN {X -125.8897,Y -20.5917,Z 139,A -174.5686,B 24.9591,C -1.4776,E1 24.8417,E2 620.9974} C_DIS
LIN {X -126.3424,Y -17.6032,Z 139,A -175.8835,B 24.9587,C -1.4839,E1 24.8412,E2 622.305} C_DIS
LIN {X -126.7461,Y -14.4212,Z 139,A -177.3511,B 24.9586,C -1.4873,E1 24.8407,E2 623.7733} C_DIS
LIN {X -127.1061,Y -10.7759,Z 139,A -179.0689,B 24.9584,C -1.4894,E1 24.8403,E2 625.4964} C_DIS
LIN {X -127.3244,Y -7.7839,Z 139,A 179.5771,B 24.9582,C -1.4935,E1 24.84,E2 626.8488} C_DIS
LIN {X -127.4741,Y -4.7434,Z 139,A 178.2159,B 24.9579,C -1.4982,E1 24.8399,E2 628.2069} C_DIS
LIN {X -127.555,Y -1.4944,Z 139,A 176.8102,B 24.9575,C -1.5054,E1 24.8398,E2 629.6038} C_DIS
LIN {X -127.557,Y 1.3285,Z 139,A 175.5066,B 24.9574,C -1.508,E1 24.8398,E2 630.9092} C_DIS
LIN {X -127.466,Y 4.9512,Z 139,A 173.8323,B 24.9572,C -1.5112,E1 24.8399,E2 632.5859} C_DIS
LIN {X -127.3138,Y 7.9555,Z 139,A 172.4786,B 24.957,C -1.5156,E1 24.8402,E2 633.9374} C_DIS
LIN {X -127.0566,Y 11.3616,Z 139,A 170.9786,B 24.9566,C -1.5222,E1 24.8405,E2 635.4307} C_DIS
LIN {X -126.7878,Y 14.0391,Z 139,A 169.7716,B 24.9564,C -1.5262,E1 24.8409,E2 636.6352} C_DIS
LIN {X -126.4283,Y 16.9742,Z 139,A 168.3775,B 24.9563,C -1.5276,E1 24.8413,E2 638.0344} C_DIS
LIN {X -125.999,Y 19.9115,Z 139,A 167.0668,B 24.956,C -1.533,E1 24.8419,E2 639.3401} C_DIS
LIN {X -125.4682,Y 23.0236,Z 139,A 165.6464,B 24.9557,C -1.5375,E1 24.8426,E2 640.7581} C_DIS
LIN {X -124.8584,Y 26.1327,Z 139,A 164.1952,B 24.9555,C -1.5408,E1 24.8434,E2 642.21} C_DIS
LIN {X -124.2994,Y 28.6664,Z 139,A 162.983,B 24.9555,C -1.5425,E1 24.8441,E2 643.4252} C_DIS
LIN {X -123.5855,Y 31.6024,Z 139,A 161.6474,B 24.9551,C -1.5479,E1 24.845,E2 644.7558} C_DIS
LIN {X -122.6523,Y 35.0565,Z 139,A 160.0256,B 24.9548,C -1.5524,E1 24.8462,E2 646.3763} C_DIS
LIN {X -121.763,Y 38.0306,Z 139,A 158.6199,B 24.9546,C -1.5563,E1 24.8474,E2 647.7807} C_DIS
LIN {X -120.9209,Y 40.6233,Z 139,A 157.3583,B 24.9545,C -1.5586,E1 24.8485,E2 649.0442} C_DIS
LIN {X -119.9054,Y 43.5291,Z 139,A 155.9911,B 24.9542,C -1.5636,E1 24.8498,E2 650.4071} C_DIS
LIN {X -118.7464,Y 46.5987,Z 139,A 154.5008,B 24.954,C -1.5675,E1 24.8513,E2 651.8965} C_DIS
LIN {X -117.4025,Y 49.8926,Z 139,A 152.896,B 24.9537,C -1.5721,E1 24.853,E2 653.4992} C_DIS
LIN {X -116.3242,Y 52.352,Z 139,A 151.6725,B 24.9535,C -1.5751,E1 24.8544,E2 654.7224} C_DIS
LIN {X -114.7905,Y 55.6385,Z 139,A 150.0488,B 24.9532,C -1.5803,E1 24.8563,E2 656.3425} C_DIS
LIN {X -113.5221,Y 58.1792,Z 139,A 148.7127,B 24.9532,C -1.5814,E1 24.858,E2 657.6832} C_DIS
LIN {X -111.5493,Y 61.8807,Z 139,A 146.7651,B 24.953,C -1.5841,E1 24.8606,E2 659.6346} C_DIS
LIN {X -109.3678,Y 65.6605,Z 139,A 144.8852,B 24.9524,C -1.5935,E1 24.8632,E2 661.5019} C_DIS
LIN {X -107.3545,Y 68.9019,Z 139,A 143.0793,B 24.9524,C -1.5943,E1 24.8659,E2 663.3152} C_DIS
LIN {X -104.9775,Y 72.4727,Z 139,A 141.1224,B 24.9521,C -1.5983,E1 24.869,E2 665.2721} C_DIS
LIN {X -102.5752,Y 75.8349,Z 139,A 139.2132,B 24.952,C -1.6011,E1 24.8721,E2 667.1841} C_DIS
LIN {X -99.9349,Y 79.2811,Z 139,A 137.2775,B 24.9516,C -1.607,E1 24.8755,E2 669.1147} C_DIS
LIN {X -97.1671,Y 82.6499,Z 139,A 135.3586,B 24.9512,C -1.614,E1 24.8789,E2 671.0259} C_DIS
LIN {X -94.3755,Y 85.8238,Z 139,A 133.4247,B 24.951,C -1.6173,E1 24.8825,E2 672.9605} C_DIS
LIN {X -91.3766,Y 89.0108,Z 139,A 131.4285,B 24.9508,C -1.6208,E1 24.8863,E2 674.957} C_DIS
LIN {X -88.4333,Y 91.9357,Z 139,A 129.5156,B 24.9506,C -1.6231,E1 24.8902,E2 676.8725} C_DIS
LIN {X -85.3329,Y 94.82,Z 139,A 127.6117,B 24.9504,C -1.6275,E1 24.8941,E2 678.7736} C_DIS
LIN {X -81.873,Y 97.8227,Z 139,A 125.5958,B 24.95,C -1.6341,E1 24.8983,E2 680.7816} C_DIS
LIN {X -78.4909,Y 100.5574,Z 139,A 123.6118,B 24.9498,C -1.637,E1 24.9027,E2 682.7661} C_DIS
LIN {X -75.1928,Y 103.0468,Z 139,A 121.7225,B 24.9496,C -1.6394,E1 24.9069,E2 684.6565} C_DIS
LIN {X -71.6882,Y 105.5145,Z 139,A 119.8078,B 24.9494,C -1.6438,E1 24.9113,E2 686.5672} C_DIS
LIN {X -67.8968,Y 107.9932,Z 139,A 117.7899,B 24.9491,C -1.6485,E1 24.916,E2 688.5803} C_DIS
LIN {X -64.2618,Y 110.1955,Z 139,A 115.9237,B 24.9487,C -1.654,E1 24.9205,E2 690.439} C_DIS
LIN {X -60.7302,Y 112.1805,Z 139,A 113.9962,B 24.9488,C -1.6522,E1 24.9252,E2 692.3764} C_DIS
LIN {X -57.6088,Y 113.8125,Z 139,A 112.5351,B 24.9483,C -1.6605,E1 24.9288,E2 693.8217} C_DIS
LIN {X -54.2652,Y 115.4465,Z 139,A 110.8768,B 24.9481,C -1.6638,E1 24.933,E2 695.4765} C_DIS
LIN {X -51.7226,Y 116.6058,Z 139,A 109.5999,B 24.9481,C -1.6647,E1 24.9362,E2 696.7544} C_DIS
LIN {X -48.4756,Y 117.9943,Z 139,A 108.0298,B 24.9479,C -1.6677,E1 24.9403,E2 698.3208} C_DIS
LIN {X -45.854,Y 119.0359,Z 139,A 106.7311,B 24.9479,C -1.668,E1 24.9436,E2 699.6217} C_DIS
LIN {X -42.9572,Y 120.1115,Z 139,A 105.3757,B 24.9477,C -1.6714,E1 24.9472,E2 700.9718} C_DIS
LIN {X -39.7537,Y 121.2105,Z 139,A 103.8477,B 24.9476,C -1.6729,E1 24.9512,E2 702.499} C_DIS
LIN {X -36.5878,Y 122.2045,Z 139,A 102.3547,B 24.9475,C -1.6745,E1 24.9552,E2 703.9909} C_DIS
LIN {X -34.0448,Y 122.9352,Z 139,A 101.1795,B 24.9473,C -1.6764,E1 24.9584,E2 705.1634} C_DIS
LIN {X -31.009,Y 123.7361,Z 139,A 99.7764,B 24.9473,C -1.6782,E1 24.9622,E2 706.5643} C_DIS
LIN {X -27.8122,Y 124.4945,Z 139,A 98.2958,B 24.9472,C -1.6793,E1 24.9662,E2 708.0441} C_DIS
LIN {X -24.6938,Y 125.1512,Z 139,A 96.8457,B 24.9472,C -1.6796,E1 24.9702,E2 709.4952} C_DIS
LIN {X -22.2616,Y 125.6046,Z 139,A 95.678,B 24.9472,C -1.6778,E1 24.9734,E2 710.6684} C_DIS
LIN {X -19.0227,Y 126.1366,Z 139,A 94.281,B 24.9469,C -1.6826,E1 24.9772,E2 712.0554} C_DIS
LIN {X -15.8854,Y 126.571,Z 139,A 92.6802,B 24.9474,C -1.6749,E1 24.9817,E2 713.6756} C_DIS
LIN {X -12.1274,Y 126.9843,Z 139,A 91.1299,B 24.9469,C -1.6829,E1 24.9859,E2 715.2078} C_DIS
LIN {X -8.5644,Y 127.2763,Z 139,A 89.4975,B 24.9469,C -1.6823,E1 24.9905,E2 716.8423} C_DIS
LIN {X -5.0353,Y 127.4628,Z 139,A 87.9466,B 24.9469,C -1.6847,E1 24.9948,E2 718.388} C_DIS
LIN {X -1.8561,Y 127.549,Z 139,A 86.5254,B 24.9468,C -1.6854,E1 24.9988,E2 719.8076} C_DIS
LIN {X 0.9343,Y 127.559,Z 139,A 85.2761,B 24.9468,C -1.6858,E1 25.0023,E2 721.0557} C_DIS
LIN {X 3.7744,Y 127.5065,Z 139,A 83.9472,B 24.9468,C -1.6834,E1 25.006,E2 722.3901} C_DIS
LIN {X 7.924,Y 127.3158,Z 139,A 82.0462,B 24.947,C -1.6817,E1 25.0113,E2 724.2945} C_DIS
LIN {X 11.4525,Y 127.049,Z 139,A 80.3589,B 24.9473,C -1.6768,E1 25.016,E2 725.9925} C_DIS
LIN {X 15.2314,Y 126.6495,Z 139,A 78.7511,B 24.947,C -1.6814,E1 25.0204,E2 727.5884} C_DIS
LIN {X 18.5028,Y 126.2138,Z 139,A 77.3581,B 24.9468,C -1.6853,E1 25.0243,E2 728.9707} C_DIS
LIN {X 21.6888,Y 125.7066,Z 139,A 75.8924,B 24.9468,C -1.684,E1 25.0283,E2 730.4381} C_DIS
LIN {X 24.2628,Y 125.2336,Z 139,A 74.7453,B 24.9468,C -1.6849,E1 25.0314,E2 731.5817} C_DIS
LIN {X 27.1239,Y 124.645,Z 139,A 73.3444,B 24.9471,C -1.6799,E1 25.0353,E2 732.9927} C_DIS
LIN {X 30.236,Y 123.9272,Z 139,A 71.927,B 24.9471,C -1.6799,E1 25.0391,E2 734.408} C_DIS
LIN {X 33.1334,Y 123.1839,Z 139,A 70.5732,B 24.9471,C -1.6786,E1 25.0428,E2 735.763} C_DIS
LIN {X 36.4146,Y 122.2552,Z 139,A 69.1078,B 24.9471,C -1.6807,E1 25.0467,E2 737.2208} C_DIS
LIN {X 39.5065,Y 121.2921,Z 139,A 67.6396,B 24.9471,C -1.6789,E1 25.0506,E2 738.6907} C_DIS
LIN {X 42.3358,Y 120.3329,Z 139,A 66.2975,B 24.9473,C -1.6777,E1 25.0542,E2 740.0329} C_DIS
LIN {X 45.1962,Y 119.2876,Z 139,A 64.9052,B 24.9474,C -1.6752,E1 25.0578,E2 741.4282} C_DIS
LIN {X 48.1972,Y 118.1072,Z 139,A 63.4651,B 24.9474,C -1.6741,E1 25.0616,E2 742.8677} C_DIS
LIN {X 50.9373,Y 116.9508,Z 139,A 62.1033,B 24.9477,C -1.6713,E1 25.0651,E2 744.2328} C_DIS
LIN {X 54.1411,Y 115.5039,Z 139,A 60.5831,B 24.9476,C -1.6723,E1 25.0689,E2 745.7467} C_DIS
LIN {X 57.1116,Y 114.0649,Z 139,A 59.0954,B 24.9477,C -1.6702,E1 25.0726,E2 747.2355} C_DIS
LIN {X 59.6016,Y 112.7818,Z 139,A 57.7974,B 24.948,C -1.6665,E1 25.0759,E2 748.5386} C_DIS
LIN {X 62.8549,Y 111.004,Z 139,A 56.0316,B 24.9484,C -1.6591,E1 25.0802,E2 750.3167} C_DIS
LIN {X 66.3362,Y 108.9592,Z 139,A 54.327,B 24.9483,C -1.6618,E1 25.0843,E2 752.0097} C_DIS
LIN {X 69.8044,Y 106.7706,Z 139,A 52.3782,B 24.9488,C -1.6534,E1 25.0889,E2 753.9719} C_DIS
LIN {X 73.4055,Y 104.3269,Z 139,A 50.4804,B 24.9488,C -1.653,E1 25.0932,E2 755.8642} C_DIS
LIN {X 76.4937,Y 102.0848,Z 139,A 48.7625,B 24.949,C -1.6497,E1 25.0971,E2 757.5837} C_DIS
LIN {X 79.7626,Y 99.5517,Z 139,A 47.0189,B 24.9489,C -1.652,E1 25.1009,E2 759.3154} C_DIS
LIN {X 82.2883,Y 97.4743,Z 139,A 45.5155,B 24.9491,C -1.6474,E1 25.1041,E2 760.824} C_DIS
LIN {X 85.3447,Y 94.8094,Z 139,A 43.7391,B 24.9492,C -1.646,E1 25.1078,E2 762.5967} C_DIS
LIN {X 88.1233,Y 92.2319,Z 139,A 41.959,B 24.9497,C -1.6384,E1 25.1115,E2 764.3872} C_DIS
LIN {X 91.311,Y 89.0778,Z 139,A 40.0041,B 24.9497,C -1.6371,E1 25.1153,E2 766.3371} C_DIS
LIN {X 94.1315,Y 86.0919,Z 139,A 38.1151,B 24.9502,C -1.6306,E1 25.1189,E2 768.233} C_DIS
LIN {X 96.9248,Y 82.9349,Z 139,A 36.2012,B 24.9505,C -1.6251,E1 25.1224,E2 770.1512} C_DIS
LIN {X 99.6195,Y 79.6774,Z 139,A 34.3084,B 24.9508,C -1.6208,E1 25.1258,E2 772.0454} C_DIS
LIN {X 102.0704,Y 76.5131,Z 139,A 32.598,B 24.9508,C -1.6208,E1 25.1286,E2 773.7476} C_DIS
LIN {X 104.4777,Y 73.1917,Z 139,A 30.6653,B 24.9513,C -1.6115,E1 25.1318,E2 775.693} C_DIS
LIN {X 106.8283,Y 69.7155,Z 139,A 28.803,B 24.9516,C -1.6077,E1 25.1347,E2 777.555} C_DIS
LIN {X 109.207,Y 65.9264,Z 139,A 26.8959,B 24.9516,C -1.6076,E1 25.1375,E2 779.4527} C_DIS
LIN {X 111.1549,Y 62.5863,Z 139,A 25.1307,B 24.952,C -1.6013,E1 25.1399,E2 781.2235} C_DIS
LIN {X 113.0705,Y 59.0518,Z 139,A 23.3963,B 24.952,C -1.6,E1 25.1422,E2 782.9519} C_DIS
LIN {X 114.7551,Y 55.7126,Z 139,A 21.7545,B 24.9522,C -1.5971,E1 25.1442,E2 784.5917} C_DIS
LIN {X 115.9042,Y 53.2754,Z 139,A 20.5074,B 24.9525,C -1.5918,E1 25.1457,E2 785.8447} C_DIS
LIN {X 117.2041,Y 50.3515,Z 139,A 19.0819,B 24.9527,C -1.5881,E1 25.1473,E2 787.271} C_DIS
LIN {X 118.4696,Y 47.2983,Z 139,A 17.6653,B 24.9527,C -1.5873,E1 25.1488,E2 788.6818} C_DIS
LIN {X 119.6001,Y 44.3619,Z 139,A 16.2651,B 24.953,C -1.5837,E1 25.1502,E2 790.0826} C_DIS
LIN {X 120.705,Y 41.2628,Z 139,A 14.7812,B 24.9533,C -1.5789,E1 25.1515,E2 791.5695} C_DIS
LIN {X 121.7356,Y 38.1182,Z 139,A 13.3079,B 24.9535,C -1.575,E1 25.1528,E2 793.0436} C_DIS
LIN {X 122.6401,Y 35.1003,Z 139,A 11.9044,B 24.9537,C -1.5712,E1 25.1539,E2 794.448} C_DIS
LIN {X 123.3314,Y 32.5804,Z 139,A 10.7593,B 24.9539,C -1.5691,E1 25.1547,E2 795.5916} C_DIS
LIN {X 124.1079,Y 29.4862,Z 139,A 9.3317,B 24.9541,C -1.5648,E1 25.1557,E2 797.021} C_DIS
LIN {X 124.7654,Y 26.5664,Z 139,A 7.953,B 24.9545,C -1.5588,E1 25.1565,E2 798.4059} C_DIS
LIN {X 125.6184,Y 22.1845,Z 139,A 6.002,B 24.9547,C -1.5552,E1 25.1575,E2 800.3539} C_DIS
LIN {X 126.1537,Y 18.9124,Z 139,A 4.5312,B 24.9549,C -1.5514,E1 25.1582,E2 801.8251} C_DIS
LIN {X 126.4986,Y 16.4376,Z 139,A 3.3427,B 24.9553,C -1.5443,E1 25.1586,E2 803.0232} C_DIS
LIN {X 126.8622,Y 13.3474,Z 139,A 1.9985,B 24.9554,C -1.5425,E1 25.159,E2 804.3636} C_DIS
LIN {X 127.1203,Y 10.6076,Z 139,A 0.7954,B 24.9556,C -1.5403,E1 25.1593,E2 805.565} C_DIS
LIN {X 127.3651,Y 7.123,Z 139,A -0.7584,B 24.9558,C -1.5359,E1 25.1596,E2 807.1199} C_DIS
LIN {X 127.5316,Y 2.8734,Z 139,A -2.7898,B 24.9565,C -1.5232,E1 25.1598,E2 809.1689} C_DIS
LIN {X 127.5599,Y -0.8146,Z 139,A -4.3739,B 24.9566,C -1.5216,E1 25.1598,E2 810.7474} C_DIS
LIN {X 127.4462,Y -5.4589,Z 139,A -6.384,B 24.9568,C -1.5188,E1 25.1596,E2 812.7523} C_DIS
LIN {X 127.2329,Y -9.1594,Z 139,A -8.0806,B 24.9572,C -1.5116,E1 25.1593,E2 814.4557} C_DIS
LIN {X 126.9084,Y -12.918,Z 139,A -9.7149,B 24.9573,C -1.5092,E1 25.1589,E2 816.0861} C_DIS
LIN {X 126.6411,Y -15.3017,Z 139,A -10.7841,B 24.9575,C -1.5061,E1 25.1585,E2 817.1562} C_DIS
LIN {X 126.2032,Y -18.5769,Z 139,A -12.2468,B 24.9577,C -1.5023,E1 25.158,E2 818.6193} C_DIS
LIN {X 125.7819,Y -21.2373,Z 139,A -13.5047,B 24.9581,C -1.4958,E1 25.1574,E2 819.885} C_DIS
LIN {X 125.2302,Y -24.2809,Z 139,A -14.8826,B 24.9583,C -1.4919,E1 25.1567,E2 821.2642} C_DIS
LIN {X 124.5713,Y -27.4653,Z 139,A -16.3094,B 24.9585,C -1.4889,E1 25.1559,E2 822.6898} C_DIS
LIN {X 123.8987,Y -30.3542,Z 139,A -17.6455,B 24.9587,C -1.4843,E1 25.155,E2 824.0288} C_DIS
LIN {X 123.1125,Y -33.4011,Z 139,A -19.0059,B 24.9588,C -1.4825,E1 25.154,E2 825.3856} C_DIS
LIN {X 122.2501,Y -36.432,Z 139,A -20.4204,B 24.9591,C -1.478,E1 25.1529,E2 826.8027} C_DIS
LIN {X 121.4209,Y -39.1032,Z 139,A -21.7315,B 24.9595,C -1.4711,E1 25.1518,E2 828.1226} C_DIS
LIN {X 120.44,Y -42.027,Z 139,A -23.099,B 24.9596,C -1.4676,E1 25.1506,E2 829.4905} C_DIS
LIN {X 119.1806,Y -45.4819,Z 139,A -24.7102,B 24.9598,C -1.4645,E1 25.149,E2 831.1002} C_DIS
LIN {X 118.0324,Y -48.3827,Z 139,A -26.1042,B 24.96,C -1.4605,E1 25.1475,E2 832.4959} C_DIS
LIN {X 116.7889,Y -51.3117,Z 139,A -27.5228,B 24.9603,C -1.4566,E1 25.146,E2 833.9159} C_DIS
LIN {X 115.4465,Y -54.2652,Z 139,A -28.9743,B 24.9605,C -1.4524,E1 25.1443,E2 835.3695} C_DIS
LIN {X 114.2182,Y -56.8008,Z 139,A -30.2642,B 24.9608,C -1.4473,E1 25.1427,E2 836.6645} C_DIS
LIN {X 112.2594,Y -60.5833,Z 139,A -32.2219,B 24.9612,C -1.4392,E1 25.1401,E2 838.6311} C_DIS
LIN {X 110.1955,Y -64.2618,Z 139,A -34.1369,B 24.9616,C -1.4325,E1 25.1375,E2 840.552} C_DIS
LIN {X 107.9976,Y -67.8898,Z 139,A -36.0331,B 24.9618,C -1.4274,E1 25.1347,E2 842.4505} C_DIS
LIN {X 105.608,Y -71.55,Z 139,A -37.9189,B 24.9619,C -1.4258,E1 25.1318,E2 844.3306} C_DIS
LIN {X 103.2092,Y -74.9689,Z 139,A -39.7697,B 24.9621,C -1.4218,E1 25.1288,E2 846.1818} C_DIS
LIN {X 100.9432,Y -77.9933,Z 139,A -41.5307,B 24.9626,C -1.4138,E1 25.1258,E2 847.9533} C_DIS
LIN {X 98.196,Y -81.4248,Z 139,A -43.4307,B 24.9626,C -1.4124,E1 25.1224,E2 849.8479} C_DIS
LIN {X 95.8666,Y -84.1557,Z 139,A -44.9908,B 24.9627,C -1.4108,E1 25.1196,E2 851.4046} C_DIS
LIN {X 93.3748,Y -86.9115,Z 139,A -46.717,B 24.9631,C -1.4035,E1 25.1163,E2 853.1404} C_DIS
LIN {X 90.4959,Y -89.9051,Z 139,A -48.5714,B 24.9633,C -1.3994,E1 25.1127,E2 854.9965} C_DIS
LIN {X 87.8365,Y -92.506,Z 139,A -50.2237,B 24.9635,C -1.3963,E1 25.1094,E2 856.6494} C_DIS
LIN {X 84.817,Y -95.282,Z 139,A -52.1339,B 24.9639,C -1.3884,E1 25.1054,E2 858.5705} C_DIS
LIN {X 81.5058,Y -98.1289,Z 139,A -54.0562,B 24.964,C -1.3859,E1 25.1013,E2 860.4912} C_DIS
LIN {X 78.3091,Y -100.6984,Z 139,A -55.8923,B 24.9642,C -1.3821,E1 25.0973,E2 862.3295} C_DIS
LIN {X 75.0824,Y -103.1269,Z 139,A -57.7173,B 24.9644,C -1.3777,E1 25.0932,E2 864.1585} C_DIS
LIN {X 71.2903,Y -105.7838,Z 139,A -59.7413,B 24.9645,C -1.3763,E1 25.0885,E2 866.1788} C_DIS
LIN {X 67.7426,Y -108.0905,Z 139,A -61.5498,B 24.9645,C -1.3772,E1 25.0843,E2 867.9792} C_DIS
LIN {X 64.5148,Y -110.0469,Z 139,A -63.3357,B 24.9649,C -1.3694,E1 25.08,E2 869.7781} C_DIS
LIN {X 60.7302,Y -112.1805,Z 139,A -65.3316,B 24.9652,C -1.3636,E1 25.0751,E2 871.7818} C_DIS
LIN {X 57.6201,Y -113.8067,Z 139,A -66.7501,B 24.9649,C -1.369,E1 25.0716,E2 873.1836} C_DIS
LIN {X 54.6883,Y -115.2444,Z 139,A -68.2482,B 24.9651,C -1.365,E1 25.0678,E2 874.6873} C_DIS
LIN {X 51.714,Y -116.6096,Z 139,A -69.6557,B 24.9651,C -1.3659,E1 25.0642,E2 876.0891} C_DIS
LIN {X 48.6914,Y -117.9042,Z 139,A -71.1595,B 24.9652,C -1.3623,E1 25.0604,E2 877.5979} C_DIS
LIN {X 45.8985,Y -119.0186,Z 139,A -72.467,B 24.9652,C -1.3626,E1 25.057,E2 878.9018} C_DIS
LIN {X 43.0397,Y -120.0818,Z 139,A -73.8688,B 24.9654,C -1.3591,E1 25.0533,E2 880.3089} C_DIS
LIN {X 39.6035,Y -121.2605,Z 139,A -75.4784,B 24.9654,C -1.3582,E1 25.049,E2 881.9177} C_DIS
LIN {X 37.138,Y -122.0362,Z 139,A -76.6791,B 24.9656,C -1.3548,E1 25.0458,E2 883.1242} C_DIS
LIN {X 33.6769,Y -123.0381,Z 139,A -78.2393,B 24.9656,C -1.3559,E1 25.0416,E2 884.6792} C_DIS
LIN {X 30.6803,Y -123.8195,Z 139,A -79.6298,B 24.9656,C -1.3545,E1 25.0379,E2 886.071} C_DIS
LIN {X 28.2303,Y -124.399,Z 139,A -80.7972,B 24.9658,C -1.3516,E1 25.0347,E2 887.2436} C_DIS
LIN {X 25.0717,Y -125.0743,Z 139,A -82.1682,B 24.9656,C -1.3543,E1 25.0309,E2 888.6065} C_DIS
LIN {X 22.3044,Y -125.5969,Z 139,A -83.5307,B 24.9659,C -1.3483,E1 25.0272,E2 889.9816} C_DIS
LIN {X 18.8745,Y -126.1596,Z 139,A -85.0054,B 24.9658,C -1.3515,E1 25.0231,E2 891.4474} C_DIS
LIN {X 15.8854,Y -126.571,Z 139,A -86.4598,B 24.9661,C -1.3456,E1 25.0191,E2 892.9144} C_DIS
LIN {X 12.2785,Y -126.9698,Z 139,A -88.0031,B 24.9659,C -1.3491,E1 25.0148,E2 894.4486} C_DIS
LIN {X 9.0454,Y -127.2412,Z 139,A -89.4935,B 24.966,C -1.3467,E1 25.0106,E2 895.9439} C_DIS
LIN {X 5.9449,Y -127.4244,Z 139,A -90.8029,B 24.9658,C -1.3504,E1 25.007,E2 897.244} C_DIS
LIN {X 3.4372,Y -127.5159,Z 139,A -92.0231,B 24.9661,C -1.3454,E1 25.0036,E2 898.4758} C_DIS
LIN {X 0.903,Y -127.5582,Z 139,A -92.8334,B 24.9653,C -1.3614,E1 25.0014,E2 899.248} C_DIS
Enddeposition()
LIN {X 0.903,Y -127.5582,Z 139,A -92.8334,B 24.9653,C -1.3614,E1 25.0014,E2 899.248} C_DIS
Startdeposition()
$VEL.CP = VEL_PRINT
LIN {X 3.1927,Y -126.5433,Z 139,A -91.4315,B 24.9634,C -1.397,E1 25.0056,E2 897.7619} C_DIS
LIN {X 7.0361,Y -126.3893,Z 139,A -89.5936,B 24.9632,C -1.4025,E1 25.0107,E2 895.9116} C_DIS
LIN {X 11.007,Y -126.1041,Z 139,A -87.8319,B 24.9632,C -1.4014,E1 25.0156,E2 894.1535} C_DIS
LIN {X 15.0322,Y -125.6873,Z 139,A -86.0987,B 24.9634,C -1.3976,E1 25.0204,E2 892.4306} C_DIS
LIN {X 18.9833,Y -125.152,Z 139,A -84.2495,B 24.9632,C -1.4011,E1 25.0255,E2 890.5748} C_DIS
LIN {X 22.4672,Y -124.5732,Z 139,A -82.6679,B 24.9632,C -1.4015,E1 25.0299,E2 888.9939} C_DIS
LIN {X 26.5505,Y -123.7672,Z 139,A -80.8208,B 24.9632,C -1.4013,E1 25.0349,E2 887.1495} C_DIS
LIN {X 29.7506,Y -123.0371,Z 139,A -79.3472,B 24.9632,C -1.4021,E1 25.0389,E2 885.676} C_DIS
LIN {X 32.8422,Y -122.2483,Z 139,A -77.5705,B 24.9622,C -1.4206,E1 25.0438,E2 883.8584} C_DIS
LIN {X 36.1312,Y -121.3181,Z 139,A -76.2471,B 24.9627,C -1.411,E1 25.0473,E2 882.5601} C_DIS
LIN {X 43.58,Y -118.8457,Z 139,A -72.8296,B 24.9628,C -1.4086,E1 25.0563,E2 879.155} C_DIS
LIN {X 46.2737,Y -117.8224,Z 139,A -71.3939,B 24.9624,C -1.4171,E1 25.0601,E2 877.7022} C_DIS
LIN {X 49.4819,Y -116.5131,Z 139,A -69.9835,B 24.9627,C -1.4113,E1 25.0637,E2 876.3088} C_DIS
LIN {X 53.1875,Y -114.8663,Z 139,A -68.1277,B 24.9625,C -1.4153,E1 25.0684,E2 874.4483} C_DIS
LIN {X 56.1814,Y -113.4322,Z 139,A -66.6154,B 24.9623,C -1.4183,E1 25.0722,E2 872.9329} C_DIS
LIN {X 60.0061,Y -111.4582,Z 139,A -64.6291,B 24.962,C -1.4236,E1 25.0771,E2 870.9397} C_DIS
LIN {X 63.707,Y -109.3854,Z 139,A -62.6888,B 24.9618,C -1.4281,E1 25.0819,E2 868.9944} C_DIS
LIN {X 67.1235,Y -107.3227,Z 139,A -60.5135,B 24.9606,C -1.4508,E1 25.0871,E2 866.7725} C_DIS
LIN {X 70.4431,Y -105.1734,Z 139,A -58.5114,B 24.9598,C -1.4655,E1 25.0918,E2 864.7423} C_DIS
LIN {X 74.5963,Y -102.2698,Z 139,A -57.1027,B 24.962,C -1.4242,E1 25.0948,E2 863.4361} C_DIS
LIN {X 78.9656,Y -98.9348,Z 139,A -54.3991,B 24.9611,C -1.4408,E1 25.1008,E2 860.7032} C_DIS
LIN {X 82.2417,Y -96.2292,Z 139,A -52.3986,B 24.9607,C -1.4493,E1 25.1051,E2 858.6905} C_DIS
LIN {X 85.4855,Y -93.3591,Z 139,A -50.198,B 24.9597,C -1.4665,E1 25.1098,E2 856.458} C_DIS
LIN {X 88.0296,Y -90.9639,Z 139,A -48.722,B 24.9598,C -1.4649,E1 25.1127,E2 854.9921} C_DIS
LIN {X 91.8483,Y -87.107,Z 139,A -46.4487,B 24.96,C -1.4614,E1 25.1171,E2 852.7367} C_DIS
LIN {X 94.7427,Y -83.9492,Z 139,A -44.1127,B 24.9586,C -1.4874,E1 25.1215,E2 850.3499} C_DIS
LIN {X 97.4765,Y -80.7587,Z 139,A -42.8237,B 24.9601,C -1.4602,E1 25.1237,E2 849.1309} C_DIS
LIN {X 99.6533,Y -78.0568,Z 139,A -40.8249,B 24.9586,C -1.487,E1 25.1273,E2 847.0783} C_DIS
LIN {X 101.7199,Y -75.3446,Z 139,A -39.7676,B 24.9598,C -1.4657,E1 25.1289,E2 846.0762} C_DIS
LIN {X 104.0732,Y -72.0589,Z 139,A -37.7072,B 24.9588,C -1.483,E1 25.1323,E2 843.9851} C_DIS
LIN {X 106.5177,Y -68.3933,Z 139,A -35.7297,B 24.9585,C -1.4878,E1 25.1353,E2 842.0061} C_DIS
LIN {X 108.925,Y -64.4911,Z 139,A -33.6427,B 24.9582,C -1.4945,E1 25.1384,E2 839.914} C_DIS
LIN {X 111.115,Y -60.639,Z 139,A -31.6758,B 24.9579,C -1.4985,E1 25.141,E2 837.948} C_DIS
LIN {X 112.9647,Y -57.1162,Z 139,A -30.0479,B 24.9581,C -1.4948,E1 25.1431,E2 836.3373} C_DIS
LIN {X 114.5608,Y -53.8468,Z 139,A -28.2963,B 24.9575,C -1.5054,E1 25.1452,E2 834.5703} C_DIS
LIN {X 115.871,Y -50.9658,Z 139,A -26.9772,B 24.9576,C -1.5038,E1 25.1467,E2 833.262} C_DIS
LIN {X 116.8881,Y -48.584,Z 139,A -25.7278,B 24.9572,C -1.5116,E1 25.1481,E2 832.0012} C_DIS
LIN {X 118.3942,Y -44.7903,Z 139,A -23.4985,B 24.9557,C -1.5377,E1 25.1503,E2 829.7228} C_DIS
LIN {X 119.6823,Y -41.2239,Z 139,A -22.1868,B 24.9566,C -1.5216,E1 25.1515,E2 828.4563} C_DIS
LIN {X 121.2969,Y -36.2036,Z 139,A -19.8115,B 24.9562,C -1.5286,E1 25.1535,E2 826.078} C_DIS
LIN {X 122.3451,Y -32.4793,Z 139,A -18.1345,B 24.9562,C -1.5304,E1 25.1547,E2 824.4065} C_DIS
LIN {X 123.194,Y -29.0998,Z 139,A -16.3035,B 24.955,C -1.549,E1 25.1559,E2 822.5423} C_DIS
LIN {X 123.9761,Y -25.5589,Z 139,A -14.8917,B 24.9554,C -1.5422,E1 25.1567,E2 821.1548} C_DIS
LIN {X 124.6429,Y -22.0778,Z 139,A -13.3195,B 24.9552,C -1.5457,E1 25.1575,E2 819.5833} C_DIS
LIN {X 125.2542,Y -18.2972,Z 139,A -11.5669,B 24.9548,C -1.5524,E1 25.1583,E2 817.8253} C_DIS
LIN {X 125.7305,Y -14.6698,Z 139,A -10.0181,B 24.9548,C -1.5522,E1 25.1588,E2 816.2861} C_DIS
LIN {X 126.0802,Y -11.2895,Z 139,A -8.3396,B 24.9541,C -1.5647,E1 25.1593,E2 814.5881} C_DIS
LIN {X 126.3781,Y -7.2234,Z 139,A -6.5071,B 24.9538,C -1.5701,E1 25.1596,E2 812.7538} C_DIS
LIN {X 126.5378,Y -3.3912,Z 139,A -4.8107,B 24.9536,C -1.5737,E1 25.1598,E2 811.0589} C_DIS
LIN {X 126.5816,Y 0.6907,Z 139,A -2.9975,B 24.9533,C -1.578,E1 25.1598,E2 809.2465} C_DIS
LIN {X 126.4903,Y 4.8489,Z 139,A -1.1703,B 24.9532,C -1.5812,E1 25.1596,E2 807.4225} C_DIS
LIN {X 126.2861,Y 8.6821,Z 139,A 0.6119,B 24.9527,C -1.5893,E1 25.1593,E2 805.632} C_DIS
LIN {X 125.999,Y 12.1463,Z 139,A 2.1258,B 24.9526,C -1.5913,E1 25.1589,E2 804.1223} C_DIS
LIN {X 125.5505,Y 16.1381,Z 139,A 4.0115,B 24.952,C -1.6007,E1 25.1583,E2 802.2255} C_DIS
LIN {X 124.9127,Y 20.4982,Z 139,A 5.9406,B 24.9518,C -1.6037,E1 25.1575,E2 800.3008} C_DIS
LIN {X 124.291,Y 23.98,Z 139,A 7.4929,B 24.9517,C -1.6062,E1 25.1567,E2 798.7515} C_DIS
LIN {X 123.4209,Y 28.1162,Z 139,A 9.3853,B 24.9514,C -1.6112,E1 25.1556,E2 796.8583} C_DIS
LIN {X 122.634,Y 31.3714,Z 139,A 10.9212,B 24.951,C -1.617,E1 25.1545,E2 795.3176} C_DIS
LIN {X 121.3149,Y 36.142,Z 139,A 13.8994,B 24.9482,C -1.663,E1 25.1521,E2 792.248} C_DIS
LIN {X 119.6467,Y 41.3265,Z 139,A 15.6744,B 24.95,C -1.634,E1 25.1506,E2 790.5514} C_DIS
LIN {X 118.0176,Y 45.7716,Z 139,A 17.7155,B 24.95,C -1.6351,E1 25.1486,E2 788.5191} C_DIS
LIN {X 116.7738,Y 48.8575,Z 139,A 19.2141,B 24.9497,C -1.6392,E1 25.147,E2 787.0192} C_DIS
LIN {X 115.3729,Y 52.0812,Z 139,A 20.7733,B 24.9495,C -1.6422,E1 25.1453,E2 785.4615} C_DIS
LIN {X 112.6719,Y 57.6912,Z 139,A 23.6201,B 24.9489,C -1.6517,E1 25.1418,E2 782.6074} C_DIS
LIN {X 110.6716,Y 61.4446,Z 139,A 25.7941,B 24.9477,C -1.67,E1 25.1388,E2 780.4016} C_DIS
LIN {X 108.3893,Y 65.3867,Z 139,A 27.6297,B 24.9481,C -1.6638,E1 25.1362,E2 778.59} C_DIS
LIN {X 106.0445,Y 69.1249,Z 139,A 29.6402,B 24.9477,C -1.6698,E1 25.1332,E2 776.5755} C_DIS
LIN {X 103.4106,Y 73.006,Z 139,A 31.6832,B 24.9477,C -1.6712,E1 25.1299,E2 774.5394} C_DIS
LIN {X 101.1461,Y 76.1127,Z 139,A 33.3652,B 24.9476,C -1.6725,E1 25.1272,E2 772.8622} C_DIS
LIN {X 98.7617,Y 79.1827,Z 139,A 35.2091,B 24.947,C -1.6812,E1 25.124,E2 771.0065} C_DIS
LIN {X 96.2263,Y 82.245,Z 139,A 36.9969,B 24.9468,C -1.6849,E1 25.1207,E2 769.2181} C_DIS
LIN {X 92.7174,Y 86.1808,Z 139,A 39.3167,B 24.9467,C -1.6869,E1 25.1164,E2 766.9038} C_DIS
LIN {X 90.4537,Y 88.5538,Z 139,A 40.8735,B 24.9462,C -1.694,E1 25.1134,E2 765.3371} C_DIS
LIN {X 85.9865,Y 92.8983,Z 139,A 43.7055,B 24.9458,C -1.7005,E1 25.1076,E2 762.5014} C_DIS
LIN {X 82.7724,Y 95.7726,Z 139,A 45.2892,B 24.9468,C -1.6856,E1 25.1044,E2 760.9591} C_DIS
LIN {X 77.7378,Y 99.9019,Z 139,A 48.5367,B 24.9454,C -1.7065,E1 25.0973,E2 757.6745} C_DIS
LIN {X 74.3606,Y 102.4409,Z 139,A 50.459,B 24.9452,C -1.7104,E1 25.0929,E2 755.7498} C_DIS
LIN {X 70.7001,Y 105.0011,Z 139,A 52.4121,B 24.9452,C -1.7104,E1 25.0885,E2 753.8035} C_DIS
LIN {X 67.8879,Y 106.8411,Z 139,A 54.0335,B 24.9447,C -1.7179,E1 25.0846,E2 752.1697} C_DIS
LIN {X 62.8258,Y 109.8935,Z 139,A 56.2724,B 24.9458,C -1.6999,E1 25.0794,E2 749.9802} C_DIS
LIN {X 58.9063,Y 112.0411,Z 139,A 58.842,B 24.9439,C -1.7303,E1 25.0729,E2 747.3462} C_DIS
LIN {X 54.4831,Y 114.2574,Z 139,A 60.7974,B 24.9446,C -1.7188,E1 25.0681,E2 745.4232} C_DIS
LIN {X 51.538,Y 115.6159,Z 139,A 62.2988,B 24.9444,C -1.7222,E1 25.0643,E2 743.9174} C_DIS
LIN {X 48.5392,Y 116.9067,Z 139,A 63.778,B 24.9444,C -1.7238,E1 25.0604,E2 742.4377} C_DIS
LIN {X 43.1214,Y 119.0116,Z 139,A 66.1199,B 24.9451,C -1.712,E1 25.0544,E2 740.1289} C_DIS
LIN {X 38.739,Y 120.5095,Z 139,A 68.4261,B 24.9443,C -1.7242,E1 25.0483,E2 737.7983} C_DIS
LIN {X 35.6266,Y 121.4659,Z 139,A 69.9389,B 24.9441,C -1.7273,E1 25.0442,E2 736.2809} C_DIS
LIN {X 32.5289,Y 122.3319,Z 139,A 71.4079,B 24.944,C -1.7289,E1 25.0402,E2 734.8104} C_DIS
LIN {X 28.6697,Y 123.2944,Z 139,A 73.3442,B 24.9435,C -1.7367,E1 25.0349,E2 732.8585} C_DIS
LIN {X 24.355,Y 124.2193,Z 139,A 75.2865,B 24.9435,C -1.7349,E1 25.0296,E2 730.9229} C_DIS
LIN {X 20.4079,Y 124.9278,Z 139,A 77.1254,B 24.9435,C -1.7367,E1 25.0246,E2 729.0815} C_DIS
LIN {X 16.4016,Y 125.5159,Z 139,A 78.8754,B 24.9437,C -1.7331,E1 25.0198,E2 727.3416} C_DIS
LIN {X 12.2957,Y 125.9846,Z 139,A 80.7127,B 24.9437,C -1.7318,E1 25.0147,E2 725.5087} C_DIS
LIN {X 8.6194,Y 126.2907,Z 139,A 82.4979,B 24.9434,C -1.7375,E1 25.0097,E2 723.7108} C_DIS
LIN {X 4.66,Y 126.4976,Z 139,A 84.2031,B 24.9437,C -1.733,E1 25.0049,E2 722.0167} C_DIS
LIN {X 0.7091,Y 126.5812,Z 139,A 85.9743,B 24.9437,C -1.7319,E1 25,E2 720.2484} C_DIS
LIN {X -3.3187,Y 126.5398,Z 139,A 87.7791,B 24.9439,C -1.7306,E1 24.995,E2 718.4466} C_DIS
LIN {X -6.985,Y 126.3918,Z 139,A 89.5672,B 24.9435,C -1.7361,E1 24.9899,E2 716.6449} C_DIS
LIN {X -10.8293,Y 126.1191,Z 139,A 91.1406,B 24.9441,C -1.7271,E1 24.9856,E2 715.0923} C_DIS
LIN {X -13.9791,Y 125.8095,Z 139,A 92.5997,B 24.9441,C -1.7276,E1 24.9816,E2 713.6312} C_DIS
LIN {X -17.7176,Y 125.3371,Z 139,A 94.3407,B 24.9441,C -1.7282,E1 24.9767,E2 711.8873} C_DIS
LIN {X -21.1267,Y 124.8078,Z 139,A 95.881,B 24.9441,C -1.7261,E1 24.9725,E2 710.3508} C_DIS
LIN {X -24.2333,Y 124.2425,Z 139,A 97.5079,B 24.9436,C -1.7344,E1 24.968,E2 708.7022} C_DIS
LIN {X -29.0356,Y 123.2094,Z 139,A 99.6363,B 24.9441,C -1.7278,E1 24.9622,E2 706.5868} C_DIS
LIN {X -32.5505,Y 122.3261,Z 139,A 101.1826,B 24.9444,C -1.7217,E1 24.9581,E2 705.0528} C_DIS
LIN {X -35.5781,Y 121.4801,Z 139,A 103.0307,B 24.9432,C -1.7404,E1 24.953,E2 703.1571} C_DIS
LIN {X -39.0936,Y 120.3951,Z 139,A 104.5384,B 24.9439,C -1.7309,E1 24.949,E2 701.6694} C_DIS
LIN {X -43.9033,Y 118.7264,Z 139,A 106.4829,B 24.9451,C -1.7108,E1 24.944,E2 699.7687} C_DIS
LIN {X -47.5206,Y 117.3244,Z 139,A 108.3926,B 24.9448,C -1.7157,E1 24.939,E2 697.8434} C_DIS
LIN {X -51.9826,Y 115.417,Z 139,A 110.5566,B 24.9451,C -1.7108,E1 24.9335,E2 695.6857} C_DIS
LIN {X -55.0945,Y 113.9654,Z 139,A 112.1077,B 24.9453,C -1.7082,E1 24.9296,E2 694.1369} C_DIS
LIN {X -57.6633,Y 112.6862,Z 139,A 113.4815,B 24.9453,C -1.7096,E1 24.9262,E2 692.7561} C_DIS
LIN {X -61.3949,Y 110.6992,Z 139,A 115.6448,B 24.9447,C -1.718,E1 24.9208,E2 690.5667} C_DIS
LIN {X -65.1106,Y 108.5558,Z 139,A 117.3921,B 24.9455,C -1.7053,E1 24.9167,E2 688.8444} C_DIS
LIN {X -68.5838,Y 106.3958,Z 139,A 119.295,B 24.9455,C -1.7041,E1 24.9122,E2 686.9382} C_DIS
LIN {X -72.1769,Y 103.9911,Z 139,A 121.2361,B 24.9459,C -1.6994,E1 24.9077,E2 685.0016} C_DIS
LIN {X -75.8119,Y 101.3719,Z 139,A 123.2694,B 24.9461,C -1.6954,E1 24.9031,E2 682.9707} C_DIS
LIN {X -79.2506,Y 98.7069,Z 139,A 125.2533,B 24.9464,C -1.6918,E1 24.8988,E2 680.9881} C_DIS
LIN {X -82.6228,Y 95.9016,Z 139,A 127.2088,B 24.9467,C -1.6859,E1 24.8946,E2 679.0391} C_DIS
LIN {X -85.9069,Y 92.9717,Z 139,A 129.2564,B 24.9469,C -1.6838,E1 24.8904,E2 676.9883} C_DIS
LIN {X -89.0839,Y 89.9317,Z 139,A 131.2443,B 24.9472,C -1.6788,E1 24.8864,E2 675.0039} C_DIS
LIN {X -92.207,Y 86.7268,Z 139,A 133.2765,B 24.9475,C -1.674,E1 24.8825,E2 672.9742} C_DIS
LIN {X -95.1346,Y 83.5056,Z 139,A 135.2851,B 24.9477,C -1.6707,E1 24.8788,E2 670.9646} C_DIS
LIN {X -97.9453,Y 80.1895,Z 139,A 137.2363,B 24.9481,C -1.6648,E1 24.8753,E2 669.0186} C_DIS
LIN {X -100.7304,Y 76.6623,Z 139,A 139.2943,B 24.9483,C -1.6603,E1 24.8718,E2 666.9614} C_DIS
LIN {X -103.3039,Y 73.1574,Z 139,A 141.2745,B 24.9486,C -1.6554,E1 24.8685,E2 664.9833} C_DIS
LIN {X -105.6354,Y 69.7483,Z 139,A 143.1505,B 24.949,C -1.6504,E1 24.8656,E2 663.1098} C_DIS
LIN {X -108.0997,Y 65.8653,Z 139,A 145.4154,B 24.9488,C -1.6528,E1 24.8623,E2 660.8276} C_DIS
LIN {X -111.0226,Y 60.8084,Z 139,A 147.8322,B 24.9499,C -1.6346,E1 24.859,E2 658.4417} C_DIS
LIN {X -112.9398,Y 57.1651,Z 139,A 149.6999,B 24.9503,C -1.6292,E1 24.8566,E2 656.5768} C_DIS
LIN {X -115.4889,Y 51.8219,Z 139,A 152.4397,B 24.9506,C -1.6237,E1 24.8534,E2 653.8352} C_DIS
LIN {X -116.9088,Y 48.5343,Z 139,A 154.0911,B 24.9508,C -1.6201,E1 24.8516,E2 652.1833} C_DIS
LIN {X -118.5991,Y 44.2432,Z 139,A 156.0842,B 24.9515,C -1.6092,E1 24.8496,E2 650.2048} C_DIS
LIN {X -119.6933,Y 41.192,Z 139,A 157.5871,B 24.9517,C -1.6062,E1 24.8482,E2 648.7006} C_DIS
LIN {X -120.8124,Y 37.7899,Z 139,A 159.1797,B 24.9521,C -1.5997,E1 24.8468,E2 647.1144} C_DIS
LIN {X -121.5484,Y 35.3445,Z 139,A 160.3534,B 24.9522,C -1.5968,E1 24.8459,E2 645.9407} C_DIS
LIN {X -122.5353,Y 31.7605,Z 139,A 162.3494,B 24.9517,C -1.6057,E1 24.8445,E2 643.912} C_DIS
LIN {X -123.721,Y 26.7648,Z 139,A 164.4739,B 24.9527,C -1.589,E1 24.8432,E2 641.8146} C_DIS
LIN {X -124.5532,Y 22.579,Z 139,A 166.3637,B 24.9532,C -1.5808,E1 24.8422,E2 639.9333} C_DIS
LIN {X -125.1804,Y 18.8002,Z 139,A 168.3693,B 24.9528,C -1.5875,E1 24.8413,E2 637.8998} C_DIS
LIN {X -125.7949,Y 14.1152,Z 139,A 170.4454,B 24.9534,C -1.5776,E1 24.8406,E2 635.8348} C_DIS
LIN {X -126.2048,Y 9.7964,Z 139,A 172.2972,B 24.954,C -1.5661,E1 24.8402,E2 633.9994} C_DIS
LIN {X -126.431,Y 6.206,Z 139,A 173.9382,B 24.9543,C -1.5613,E1 24.8399,E2 632.36} C_DIS
LIN {X -126.5635,Y 2.2374,Z 139,A 175.7149,B 24.9547,C -1.5544,E1 24.8398,E2 630.5889} C_DIS
LIN {X -126.58,Y -0.9664,Z 139,A 177.0394,B 24.9553,C -1.544,E1 24.8398,E2 629.2815} C_DIS
LIN {X -126.5277,Y -3.753,Z 139,A 178.3894,B 24.9553,C -1.5439,E1 24.8398,E2 627.9235} C_DIS
LIN {X -126.3851,Y -7.1096,Z 139,A -179.8889,B 24.9551,C -1.548,E1 24.8401,E2 626.1815} C_DIS
LIN {X -126.1234,Y -10.7782,Z 139,A -178.4267,B 24.9559,C -1.5334,E1 24.8405,E2 624.7454} C_DIS
LIN {X -125.8252,Y -13.8336,Z 139,A -176.9863,B 24.9561,C -1.5312,E1 24.8409,E2 623.3016} C_DIS
LIN {X -125.4131,Y -17.1851,Z 139,A -175.3373,B 24.9561,C -1.5317,E1 24.8415,E2 621.6415} C_DIS
LIN {X -124.7172,Y -21.6627,Z 139,A -173.4468,B 24.9568,C -1.5178,E1 24.8423,E2 619.7728} C_DIS
LIN {X -123.027,Y -29.7924,Z 139,A -169.9807,B 24.9583,C -1.4925,E1 24.8443,E2 616.3466} C_DIS
LIN {X -121.685,Y -34.8782,Z 139,A -167.1462,B 24.9575,C -1.5057,E1 24.8464,E2 613.4642} C_DIS
LIN {X -120.627,Y -38.3711,Z 139,A -165.5038,B 24.9578,C -1.5003,E1 24.8477,E2 611.8253} C_DIS
LIN {X -119.5133,Y -41.7112,Z 139,A -163.8693,B 24.958,C -1.4973,E1 24.8492,E2 610.1886} C_DIS
LIN {X -117.9848,Y -45.8559,Z 139,A -161.8547,B 24.9583,C -1.492,E1 24.8512,E2 608.1753} C_DIS
LIN {X -116.6487,Y -49.157,Z 139,A -160.2831,B 24.9587,C -1.4854,E1 24.8529,E2 606.6107} C_DIS
LIN {X -115.2897,Y -52.2671,Z 139,A -158.7604,B 24.959,C -1.4803,E1 24.8546,E2 605.0919} C_DIS
LIN {X -113.8374,Y -55.3599,Z 139,A -156.9549,B 24.9585,C -1.4878,E1 24.8568,E2 603.2586} C_DIS
LIN {X -111.7067,Y -59.5431,Z 139,A -154.9163,B 24.9591,C -1.4778,E1 24.8594,E2 601.2329} C_DIS
LIN {X -109.5929,Y -63.3485,Z 139,A -152.9956,B 24.9595,C -1.4701,E1 24.8621,E2 599.3205} C_DIS
LIN {X -107.4225,Y -66.9631,Z 139,A -151.0116,B 24.9596,C -1.4685,E1 24.865,E2 597.3302} C_DIS
LIN {X -105.0371,Y -70.6469,Z 139,A -149.0141,B 24.9599,C -1.4638,E1 24.868,E2 595.3339} C_DIS
LIN {X -102.6429,Y -74.082,Z 139,A -147.1265,B 24.9601,C -1.4586,E1 24.8711,E2 593.4493} C_DIS
LIN {X -100.2538,Y -77.2847,Z 139,A -145.2962,B 24.9603,C -1.4552,E1 24.8742,E2 591.6186} C_DIS
LIN {X -97.6669,Y -80.5288,Z 139,A -143.5345,B 24.9609,C -1.4452,E1 24.8773,E2 589.8724} C_DIS
LIN {X -95.2419,Y -83.3826,Z 139,A -141.6911,B 24.9607,C -1.4482,E1 24.8806,E2 588.0136} C_DIS
LIN {X -92.3255,Y -86.6011,Z 139,A -139.7725,B 24.9611,C -1.4415,E1 24.8843,E2 586.1024} C_DIS
LIN {X -89.4223,Y -89.5956,Z 139,A -137.8346,B 24.9611,C -1.4398,E1 24.8881,E2 584.1604} C_DIS
LIN {X -86.1237,Y -92.7706,Z 139,A -135.8277,B 24.9616,C -1.4323,E1 24.8921,E2 582.1629} C_DIS
LIN {X -82.9349,Y -95.6324,Z 139,A -133.8692,B 24.9617,C -1.4293,E1 24.8962,E2 580.2038} C_DIS
LIN {X -79.7662,Y -98.2911,Z 139,A -131.8968,B 24.9617,C -1.4305,E1 24.9005,E2 578.2211} C_DIS
LIN {X -76.3118,Y -100.9958,Z 139,A -129.9627,B 24.962,C -1.4244,E1 24.9048,E2 576.2945} C_DIS
LIN {X -72.7609,Y -103.5835,Z 139,A -127.9667,B 24.9622,C -1.4213,E1 24.9093,E2 574.2989} C_DIS
LIN {X -69.297,Y -105.9325,Z 139,A -125.1882,B 24.96,C -1.4609,E1 24.9161,E2 571.4172} C_DIS
LIN {X -63.8058,Y -109.3279,Z 139,A -123.155,B 24.9626,C -1.4135,E1 24.9207,E2 569.4905} C_DIS
LIN {X -58.9889,Y -111.9977,Z 139,A -120.6721,B 24.9628,C -1.4097,E1 24.9268,E2 567.0097} C_DIS
LIN {X -55.5584,Y -113.7395,Z 139,A -119.0238,B 24.9631,C -1.403,E1 24.9308,E2 565.3729} C_DIS
LIN {X -52.9155,Y -114.992,Z 139,A -117.6513,B 24.9631,C -1.4038,E1 24.9343,E2 563.9951} C_DIS
LIN {X -49.9316,Y -116.319,Z 139,A -115.7198,B 24.962,C -1.4241,E1 24.9394,E2 562.0107} C_DIS
LIN {X -46.294,Y -117.8145,Z 139,A -114.541,B 24.9636,C -1.3931,E1 24.9423,E2 560.903} C_DIS
Enddeposition()
END
